LIN {X 0,Y 488.723,Z 208.607,A -85,B 0,C 180,E1 -6420.22,E2 -6420.22} C_VEL
LIN {X 0,Y 488.715,Z 208.607,A -85,B 0,C 180,E1 -6423.48,E2 -6423.48} C_VEL
LIN {X 0,Y 488.671,Z 208.616,A -85,B 0,C 180,E1 -6426.352,E2 -6426.352} C_VEL
LIN {X 0,Y 488.676,Z 208.612,A -85,B 0,C 180,E1 -6429.258,E2 -6429.258} C_VEL
LIN {X 0,Y 488.654,Z 208.617,A -85,B 0,C 180,E1 -6432.531,E2 -6432.531} C_VEL
LIN {X 0,Y 488.702,Z 208.608,A -85,B 0,C 180,E1 -6435.197,E2 -6435.197} C_VEL
LIN {X 0,Y 488.648,Z 208.619,A -85,B 0,C 180,E1 -6438.578,E2 -6438.578} C_VEL
LIN {X 0,Y 488.646,Z 208.619,A -85,B 0,C 180,E1 -6441.796,E2 -6441.796} C_VEL
LIN {X 0,Y 488.678,Z 208.611,A -85,B 0,C 180,E1 -6445.061,E2 -6445.061} C_VEL
LIN {X 0,Y 488.695,Z 208.612,A -85,B 0,C 180,E1 -6448.049,E2 -6448.049} C_VEL
LIN {X 0,Y 488.667,Z 208.614,A -85,B 0,C 180,E1 -6451.32,E2 -6451.32} C_VEL
LIN {X 0,Y 488.674,Z 208.616,A -85,B 0,C 180,E1 -6453.523,E2 -6453.523} C_VEL
LIN {X 0,Y 488.675,Z 208.614,A -85,B 0,C 180,E1 -6456.253,E2 -6456.253} C_VEL
LIN {X 0,Y 488.77,Z 208.751,A -85,B 0,C 180,E1 -6459.236,E2 -6459.236} C_VEL
LIN {X 0,Y 489.525,Z 214.415,A -85,B 0,C 180,E1 -6460.5,E2 -6460.5} C_VEL
LIN {X 0,Y 489.3,Z 225.378,A -85,B 0,C 180,E1 -6462.843,E2 -6462.843} C_VEL
LIN {X 0,Y 491.728,Z 238.426,A -85,B 0,C 180,E1 -6463.139,E2 -6463.139} C_VEL
LIN {X 0,Y 490.807,Z 332.574,A -85,B 0,C 180,E1 -6464.665,E2 -6464.665} C_VEL
LIN {X 0,Y 490.602,Z 346.158,A -85,B 0,C 180,E1 -6465.057,E2 -6465.057} C_VEL
LIN {X 0,Y 490.356,Z 358.525,A -85,B 0,C 180,E1 -6465.58,E2 -6465.58} C_VEL
LIN {X 0,Y 489.939,Z 371.206,A -85,B 0,C 180,E1 -6466.309,E2 -6466.309} C_VEL
LIN {X 0,Y 489.583,Z 382.52,A -85,B 0,C 180,E1 -6467.144,E2 -6467.144} C_VEL
LIN {X 0,Y 489.305,Z 392.196,A -85,B 0,C 180,E1 -6468.033,E2 -6468.033} C_VEL
LIN {X 0,Y 488.976,Z 401.025,A -85,B 0,C 180,E1 -6469.021,E2 -6469.021} C_VEL
LIN {X 0,Y 488.645,Z 410.097,A -85,B 0,C 180,E1 -6470.27,E2 -6470.27} C_VEL
LIN {X 0,Y 488.399,Z 417.387,A -85,B 0,C 180,E1 -6471.518,E2 -6471.518} C_VEL
LIN {X 0,Y 488.261,Z 422.294,A -85,B 0,C 180,E1 -6472.556,E2 -6472.556} C_VEL
LIN {X 0,Y 488.159,Z 426.656,A -85,B 0,C 180,E1 -6473.689,E2 -6473.689} C_VEL
LIN {X 0,Y 487.975,Z 430.671,A -85,B 0,C 180,E1 -6475.042,E2 -6475.042} C_VEL
LIN {X 0,Y 488.049,Z 432.509,A -85,B 0,C 180,E1 -6475.871,E2 -6475.871} C_VEL
LIN {X 0,Y 488.018,Z 433.894,A -85,B 0,C 180,E1 -6476.697,E2 -6476.697} C_VEL
LIN {X 0,Y 488.001,Z 434.882,A -85,B 0,C 180,E1 -6477.524,E2 -6477.524} C_VEL
LIN {X 0,Y 487.897,Z 435.478,A -85,B 0,C 180,E1 -6478.349,E2 -6478.349} C_VEL
LIN {X 0,Y 487.846,Z 435.628,A -85,B 0,C 180,E1 -6479.174,E2 -6479.174} C_VEL
LIN {X 0,Y 487.853,Z 434.72,A -85,B 0,C 180,E1 -6480.825,E2 -6480.825} C_VEL
LIN {X 0,Y 487.906,Z 433.666,A -85,B 0,C 180,E1 -6481.651,E2 -6481.651} C_VEL
LIN {X 0,Y 488.031,Z 432.145,A -85,B 0,C 180,E1 -6482.476,E2 -6482.476} C_VEL
LIN {X 0,Y 488.153,Z 429.067,A -85,B 0,C 180,E1 -6483.714,E2 -6483.714} C_VEL
LIN {X 0,Y 488.245,Z 424.918,A -85,B 0,C 180,E1 -6484.954,E2 -6484.954} C_VEL
LIN {X 0,Y 488.423,Z 419.571,A -85,B 0,C 180,E1 -6486.195,E2 -6486.195} C_VEL
LIN {X 0,Y 488.576,Z 412.853,A -85,B 0,C 180,E1 -6487.438,E2 -6487.438} C_VEL
LIN {X 0,Y 488.874,Z 404.478,A -85,B 0,C 180,E1 -6488.682,E2 -6488.682} C_VEL
LIN {X 0,Y 489.2,Z 395.816,A -85,B 0,C 180,E1 -6489.718,E2 -6489.718} C_VEL
LIN {X 0,Y 489.533,Z 385.151,A -85,B 0,C 180,E1 -6490.756,E2 -6490.756} C_VEL
LIN {X 0,Y 489.943,Z 374.542,A -85,B 0,C 180,E1 -6491.585,E2 -6491.585} C_VEL
LIN {X 0,Y 490.244,Z 362.686,A -85,B 0,C 180,E1 -6492.312,E2 -6492.312} C_VEL
LIN {X 0,Y 490.576,Z 349.695,A -85,B 0,C 180,E1 -6492.912,E2 -6492.912} C_VEL
LIN {X 0,Y 490.694,Z 337.931,A -85,B 0,C 180,E1 -6493.3,E2 -6493.3} C_VEL
LIN {X 0,Y 490.842,Z 323.698,A -85,B 0,C 180,E1 -6493.586,E2 -6493.586} C_VEL
LIN {X 0,Y 491.861,Z 237.927,A -85,B 0,C 180,E1 -6495.023,E2 -6495.023} C_VEL
LIN {X 0,Y 489.611,Z 227.078,A -85,B 0,C 180,E1 -6495.32,E2 -6495.32} C_VEL
LIN {X 0,Y 490.002,Z 217.222,A -85,B 0,C 180,E1 -6497.53,E2 -6497.53} C_VEL
LIN {X 0,Y 489.355,Z 211.542,A -85,B 0,C 180,E1 -6498.888,E2 -6498.888} C_VEL
LIN {X 0,Y 488.757,Z 208.607,A -85,B 0,C 180,E1 -6499.64,E2 -6499.64} C_VEL
LIN {X 0,Y 488.727,Z 208.609,A -85,B 0,C 180,E1 -6502.847,E2 -6502.847} C_VEL
LIN {X 0,Y 488.732,Z 208.607,A -85,B 0,C 180,E1 -6505.557,E2 -6505.557} C_VEL
LIN {X 0,Y 488.749,Z 208.608,A -85,B 0,C 180,E1 -6508.328,E2 -6508.328} C_VEL
LIN {X 0,Y 488.696,Z 208.609,A -85,B 0,C 180,E1 -6511.179,E2 -6511.179} C_VEL
LIN {X 0,Y 488.736,Z 208.608,A -85,B 0,C 180,E1 -6514.112,E2 -6514.112} C_VEL
LIN {X 0,Y 488.684,Z 208.61,A -85,B 0,C 180,E1 -6517.159,E2 -6517.159} C_VEL
LIN {X 0,Y 488.723,Z 208.609,A -85,B 0,C 180,E1 -6520.344,E2 -6520.344} C_VEL
LIN {X 0,Y 488.689,Z 208.612,A -85,B 0,C 180,E1 -6523.654,E2 -6523.654} C_VEL
LIN {X 0,Y 488.683,Z 208.614,A -85,B 0,C 180,E1 -6526.344,E2 -6526.344} C_VEL
LIN {X 0,Y 488.708,Z 208.611,A -85,B 0,C 180,E1 -6529.673,E2 -6529.673} C_VEL
LIN {X 0,Y 488.675,Z 208.612,A -85,B 0,C 180,E1 -6532.84,E2 -6532.84} C_VEL
LIN {X 0,Y 488.735,Z 208.61,A -85,B 0,C 180,E1 -6535.887,E2 -6535.887} C_VEL
LIN {X 0,Y 488.697,Z 208.614,A -85,B 0,C 180,E1 -6538.82,E2 -6538.82} C_VEL
LIN {X 0,Y 488.716,Z 208.616,A -85,B 0,C 180,E1 -6541.669,E2 -6541.669} C_VEL
LIN {X 0,Y 488.748,Z 208.686,A -85,B 0,C 180,E1 -6543.871,E2 -6543.871} C_VEL
LIN {X 0,Y 490.688,Z 218.243,A -85,B 0,C 180,E1 -6545.682,E2 -6545.682} C_VEL
LIN {X 0,Y 490.806,Z 223.126,A -85,B 0,C 180,E1 -6546.539,E2 -6546.539} C_VEL
LIN {X 0,Y 490.103,Z 239.074,A -85,B 0,C 180,E1 -6549.211,E2 -6549.211} C_VEL
LIN {X 0,Y 489.482,Z 257.613,A -85,B 0,C 180,E1 -6552.234,E2 -6552.234} C_VEL
LIN {X 0,Y 489.2,Z 266.659,A -85,B 0,C 180,E1 -6553.687,E2 -6553.687} C_VEL
LIN {X 0,Y 491.59,Z 284.59,A -85,B 0,C 180,E1 -6554.091,E2 -6554.091} C_VEL
LIN {X 0,Y 490.631,Z 377.059,A -85,B 0,C 180,E1 -6555.64,E2 -6555.64} C_VEL
LIN {X 0,Y 490.339,Z 391.13,A -85,B 0,C 180,E1 -6556.055,E2 -6556.055} C_VEL
LIN {X 0,Y 489.975,Z 404.148,A -85,B 0,C 180,E1 -6556.626,E2 -6556.626} C_VEL
LIN {X 0,Y 489.605,Z 416.588,A -85,B 0,C 180,E1 -6557.355,E2 -6557.355} C_VEL
LIN {X 0,Y 489.179,Z 427.818,A -85,B 0,C 180,E1 -6558.196,E2 -6558.196} C_VEL
LIN {X 0,Y 488.867,Z 438.762,A -85,B 0,C 180,E1 -6559.228,E2 -6559.228} C_VEL
LIN {X 0,Y 488.503,Z 447.75,A -85,B 0,C 180,E1 -6560.267,E2 -6560.267} C_VEL
LIN {X 0,Y 488.3,Z 456.482,A -85,B 0,C 180,E1 -6561.516,E2 -6561.516} C_VEL
LIN {X 0,Y 488.115,Z 463.485,A -85,B 0,C 180,E1 -6562.761,E2 -6562.761} C_VEL
LIN {X 0,Y 488.008,Z 469.913,A -85,B 0,C 180,E1 -6564.213,E2 -6564.213} C_VEL
LIN {X 0,Y 487.921,Z 474.083,A -85,B 0,C 180,E1 -6565.455,E2 -6565.455} C_VEL
LIN {X 0,Y 487.969,Z 477.17,A -85,B 0,C 180,E1 -6566.696,E2 -6566.696} C_VEL
LIN {X 0,Y 487.933,Z 478.647,A -85,B 0,C 180,E1 -6567.523,E2 -6567.523} C_VEL
LIN {X 0,Y 487.892,Z 479.698,A -85,B 0,C 180,E1 -6568.348,E2 -6568.348} C_VEL
LIN {X 0,Y 487.839,Z 480.346,A -85,B 0,C 180,E1 -6569.174,E2 -6569.174} C_VEL
LIN {X 0,Y 487.829,Z 480.588,A -85,B 0,C 180,E1 -6569.999,E2 -6569.999} C_VEL
LIN {X 0,Y 487.839,Z 480.378,A -85,B 0,C 180,E1 -6570.825,E2 -6570.825} C_VEL
LIN {X 0,Y 487.892,Z 479.765,A -85,B 0,C 180,E1 -6571.65,E2 -6571.65} C_VEL
LIN {X 0,Y 487.933,Z 478.75,A -85,B 0,C 180,E1 -6572.476,E2 -6572.476} C_VEL
LIN {X 0,Y 487.968,Z 477.306,A -85,B 0,C 180,E1 -6573.302,E2 -6573.302} C_VEL
LIN {X 0,Y 487.919,Z 474.284,A -85,B 0,C 180,E1 -6574.543,E2 -6574.543} C_VEL
LIN {X 0,Y 488.001,Z 470.186,A -85,B 0,C 180,E1 -6575.785,E2 -6575.785} C_VEL
LIN {X 0,Y 488.171,Z 463.861,A -85,B 0,C 180,E1 -6577.236,E2 -6577.236} C_VEL
LIN {X 0,Y 488.301,Z 456.957,A -85,B 0,C 180,E1 -6578.483,E2 -6578.483} C_VEL
LIN {X 0,Y 488.528,Z 448.344,A -85,B 0,C 180,E1 -6579.731,E2 -6579.731} C_VEL
LIN {X 0,Y 488.853,Z 439.479,A -85,B 0,C 180,E1 -6580.771,E2 -6580.771} C_VEL
LIN {X 0,Y 489.221,Z 428.764,A -85,B 0,C 180,E1 -6581.794,E2 -6581.794} C_VEL
LIN {X 0,Y 489.581,Z 417.955,A -85,B 0,C 180,E1 -6582.623,E2 -6582.623} C_VEL
LIN {X 0,Y 490.005,Z 405.415,A -85,B 0,C 180,E1 -6583.371,E2 -6583.371} C_VEL
LIN {X 0,Y 490.327,Z 392.679,A -85,B 0,C 180,E1 -6583.943,E2 -6583.943} C_VEL
LIN {X 0,Y 490.73,Z 380.124,A -85,B 0,C 180,E1 -6584.328,E2 -6584.328} C_VEL
LIN {X 0,Y 490.899,Z 363.057,A -85,B 0,C 180,E1 -6584.641,E2 -6584.641} C_VEL
LIN {X 0,Y 491.485,Z 283.418,A -85,B 0,C 180,E1 -6585.92,E2 -6585.92} C_VEL
LIN {X 0,Y 489.262,Z 267.955,A -85,B 0,C 180,E1 -6586.266,E2 -6586.266} C_VEL
LIN {X 0,Y 489.868,Z 249.29,A -85,B 0,C 180,E1 -6589.266,E2 -6589.266} C_VEL
LIN {X 0,Y 490.552,Z 230.601,A -85,B 0,C 180,E1 -6592.311,E2 -6592.311} C_VEL
LIN {X 0,Y 490.952,Z 219.899,A -85,B 0,C 180,E1 -6594.077,E2 -6594.077} C_VEL
LIN {X 0,Y 488.78,Z 208.604,A -85,B 0,C 180,E1 -6596.125,E2 -6596.125} C_VEL
LIN {X 0,Y 488.719,Z 208.607,A -85,B 0,C 180,E1 -6599.269,E2 -6599.269} C_VEL
LIN {X 0,Y 488.7,Z 208.603,A -85,B 0,C 180,E1 -6602.146,E2 -6602.146} C_VEL
LIN {X 0,Y 488.712,Z 208.6,A -85,B 0,C 180,E1 -6605.114,E2 -6605.114} C_VEL
LIN {X 0,Y 488.67,Z 208.61,A -85,B 0,C 180,E1 -6608.2,E2 -6608.2} C_VEL
LIN {X 0,Y 488.675,Z 208.615,A -85,B 0,C 180,E1 -6611.418,E2 -6611.418} C_VEL
LIN {X 0,Y 488.695,Z 208.606,A -85,B 0,C 180,E1 -6614.802,E2 -6614.802} C_VEL
LIN {X 0,Y 488.66,Z 208.613,A -85,B 0,C 180,E1 -6617.471,E2 -6617.471} C_VEL
LIN {X 0,Y 488.686,Z 208.608,A -85,B 0,C 180,E1 -6620.744,E2 -6620.744} C_VEL
LIN {X 0,Y 488.669,Z 208.603,A -85,B 0,C 180,E1 -6623.867,E2 -6623.867} C_VEL
LIN {X 0,Y 488.727,Z 208.604,A -85,B 0,C 180,E1 -6626.876,E2 -6626.876} C_VEL
LIN {X 0,Y 488.707,Z 208.597,A -85,B 0,C 180,E1 -6629.78,E2 -6629.78} C_VEL
LIN {X 0,Y 488.689,Z 208.611,A -85,B 0,C 180,E1 -6633.078,E2 -6633.078} C_VEL
LIN {X 0,Y 488.659,Z 208.608,A -85,B 0,C 180,E1 -6636.253,E2 -6636.253} C_VEL
LIN {X 0,Y 488.737,Z 208.601,A -85,B 0,C 180,E1 -6639.176,E2 -6639.176} C_VEL
LIN {X 0,Y 488.688,Z 208.61,A -85,B 0,C 180,E1 -6642.422,E2 -6642.422} C_VEL
LIN {X 0,Y 488.741,Z 208.594,A -85,B 0,C 180,E1 -6644.999,E2 -6644.999} C_VEL
LIN {X 0,Y 488.794,Z 208.594,A -85,B 0,C 180,E1 -6648.387,E2 -6648.387} C_VEL
LIN {X 0,Y 488.768,Z 208.597,A -85,B 0,C 180,E1 -6651.733,E2 -6651.733} C_VEL
LIN {X 0,Y 488.795,Z 208.589,A -85,B 0,C 180,E1 -6654.224,E2 -6654.224} C_VEL
LIN {X 0,Y 488.94,Z 208.574,A -85,B 0,C 180,E1 -6657.529,E2 -6657.529} C_VEL
LIN {X 0,Y 488.903,Z 208.576,A -85,B 0,C 180,E1 -6660.824,E2 -6660.824} C_VEL
LIN {X 0,Y 488.94,Z 208.568,A -85,B 0,C 180,E1 -6662.472,E2 -6662.472} C_VEL
LIN {X 0,Y 488.837,Z 208.589,A -85,B 0,C 180,E1 -6665.776,E2 -6665.776} C_VEL
LIN {X 0,Y 488.806,Z 208.592,A -85,B 0,C 180,E1 -6668.267,E2 -6668.267} C_VEL
LIN {X 0,Y 488.797,Z 208.589,A -85,B 0,C 180,E1 -6671.613,E2 -6671.613} C_VEL
LIN {X 0,Y 488.754,Z 208.598,A -85,B 0,C 180,E1 -6675.001,E2 -6675.001} C_VEL
LIN {X 0,Y 488.739,Z 208.598,A -85,B 0,C 180,E1 -6678.443,E2 -6678.443} C_VEL
LIN {X 0,Y 488.7,Z 208.608,A -85,B 0,C 180,E1 -6681.071,E2 -6681.071} C_VEL
LIN {X 0,Y 488.686,Z 208.607,A -85,B 0,C 180,E1 -6683.746,E2 -6683.746} C_VEL
LIN {X 0,Y 488.784,Z 208.598,A -85,B 0,C 180,E1 -6686.944,E2 -6686.944} C_VEL
LIN {X 0,Y 488.704,Z 208.604,A -85,B 0,C 180,E1 -6690.364,E2 -6690.364} C_VEL
LIN {X 0,Y 488.73,Z 208.604,A -85,B 0,C 180,E1 -6693.485,E2 -6693.485} C_VEL
LIN {X 0,Y 488.683,Z 208.611,A -85,B 0,C 180,E1 -6696.356,E2 -6696.356} C_VEL
LIN {X 0,Y 488.697,Z 208.614,A -85,B 0,C 180,E1 -6699.255,E2 -6699.255} C_VEL
LIN {X 0,Y 488.704,Z 208.606,A -85,B 0,C 180,E1 -6701.601,E2 -6701.601} C_VEL
LIN {X 0,Y 488.709,Z 208.611,A -85,B 0,C 180,E1 -6704.802,E2 -6704.802} C_VEL
LIN {X 0,Y 488.689,Z 208.609,A -85,B 0,C 180,E1 -6707.476,E2 -6707.476} C_VEL
LIN {X 0,Y 488.731,Z 208.602,A -85,B 0,C 180,E1 -6709.678,E2 -6709.678} C_VEL
LIN {X 0,Y 488.678,Z 208.616,A -85,B 0,C 180,E1 -6712.842,E2 -6712.842} C_VEL
LIN {X 0,Y 488.733,Z 208.606,A -85,B 0,C 180,E1 -6715.889,E2 -6715.889} C_VEL
LIN {X 0,Y 488.782,Z 208.621,A -85,B 0,C 180,E1 -6718.064,E2 -6718.064} C_VEL
LIN {X 0,Y 489.044,Z 221.936,A -85,B 0,C 180,E1 -6719.712,E2 -6719.712} C_VEL
LIN {X 0,Y 491.825,Z 237.317,A -85,B 0,C 180,E1 -6720.053,E2 -6720.053} C_VEL
LIN {X 0,Y 491.789,Z 246.688,A -85,B 0,C 180,E1 -6720.193,E2 -6720.193} C_VEL
LIN {X 0,Y 491.066,Z 252.538,A -85,B 0,C 180,E1 -6720.255,E2 -6720.255} C_VEL
LIN {X 0,Y 485.39,Z 271.547,A -85,B 0,C 180,E1 -6720.34,E2 -6720.34} C_VEL
LIN {X 0,Y 484.784,Z 277.391,A -85,B 0,C 180,E1 -6720.408,E2 -6720.408} C_VEL
LIN {X 0,Y 484.329,Z 332.155,A -85,B 0,C 180,E1 -6721.242,E2 -6721.242} C_VEL
LIN {X 0,Y 484.084,Z 345.66,A -85,B 0,C 180,E1 -6721.611,E2 -6721.611} C_VEL
LIN {X 0,Y 483.812,Z 357.944,A -85,B 0,C 180,E1 -6722.125,E2 -6722.125} C_VEL
LIN {X 0,Y 483.449,Z 369.727,A -85,B 0,C 180,E1 -6722.787,E2 -6722.787} C_VEL
LIN {X 0,Y 483.011,Z 380.235,A -85,B 0,C 180,E1 -6723.539,E2 -6723.539} C_VEL
LIN {X 0,Y 482.603,Z 389.782,A -85,B 0,C 180,E1 -6724.384,E2 -6724.384} C_VEL
LIN {X 0,Y 482.225,Z 399.602,A -85,B 0,C 180,E1 -6725.459,E2 -6725.459} C_VEL
LIN {X 0,Y 481.837,Z 408.121,A -85,B 0,C 180,E1 -6726.604,E2 -6726.604} C_VEL
LIN {X 0,Y 481.49,Z 416.045,A -85,B 0,C 180,E1 -6727.924,E2 -6727.924} C_VEL
LIN {X 0,Y 481.25,Z 422.003,A -85,B 0,C 180,E1 -6729.17,E2 -6729.17} C_VEL
LIN {X 0,Y 481.061,Z 426.585,A -85,B 0,C 180,E1 -6730.367,E2 -6730.367} C_VEL
LIN {X 0,Y 480.974,Z 430.659,A -85,B 0,C 180,E1 -6731.767,E2 -6731.767} C_VEL
LIN {X 0,Y 480.818,Z 433.245,A -85,B 0,C 180,E1 -6733.003,E2 -6733.003} C_VEL
LIN {X 0,Y 480.773,Z 434.526,A -85,B 0,C 180,E1 -6733.875,E2 -6733.875} C_VEL
LIN {X 0,Y 480.791,Z 435.38,A -85,B 0,C 180,E1 -6734.746,E2 -6734.746} C_VEL
LIN {X 0,Y 480.778,Z 435.771,A -85,B 0,C 180,E1 -6735.612,E2 -6735.612} C_VEL
LIN {X 0,Y 480.753,Z 435.765,A -85,B 0,C 180,E1 -6736.474,E2 -6736.474} C_VEL
LIN {X 0,Y 480.776,Z 435.361,A -85,B 0,C 180,E1 -6737.335,E2 -6737.335} C_VEL
LIN {X 0,Y 480.847,Z 434.345,A -85,B 0,C 180,E1 -6738.314,E2 -6738.314} C_VEL
LIN {X 0,Y 480.906,Z 431.581,A -85,B 0,C 180,E1 -6739.901,E2 -6739.901} C_VEL
LIN {X 0,Y 481.007,Z 428.224,A -85,B 0,C 180,E1 -6741.176,E2 -6741.176} C_VEL
LIN {X 0,Y 481.174,Z 423.786,A -85,B 0,C 180,E1 -6742.447,E2 -6742.447} C_VEL
LIN {X 0,Y 481.388,Z 417.051,A -85,B 0,C 180,E1 -6743.925,E2 -6743.925} C_VEL
LIN {X 0,Y 481.712,Z 409.761,A -85,B 0,C 180,E1 -6745.189,E2 -6745.189} C_VEL
LIN {X 0,Y 481.991,Z 402.345,A -85,B 0,C 180,E1 -6746.239,E2 -6746.239} C_VEL
LIN {X 0,Y 482.43,Z 392.313,A -85,B 0,C 180,E1 -6747.392,E2 -6747.392} C_VEL
LIN {X 0,Y 482.82,Z 382.19,A -85,B 0,C 180,E1 -6748.333,E2 -6748.333} C_VEL
LIN {X 0,Y 483.303,Z 370.932,A -85,B 0,C 180,E1 -6749.168,E2 -6749.168} C_VEL
LIN {X 0,Y 483.676,Z 358.102,A -85,B 0,C 180,E1 -6749.897,E2 -6749.897} C_VEL
LIN {X 0,Y 483.981,Z 345.669,A -85,B 0,C 180,E1 -6750.417,E2 -6750.417} C_VEL
LIN {X 0,Y 484.228,Z 332.434,A -85,B 0,C 180,E1 -6750.781,E2 -6750.781} C_VEL
LIN {X 0,Y 484.882,Z 237.942,A -85,B 0,C 180,E1 -6752.207,E2 -6752.207} C_VEL
LIN {X 0,Y 482,Z 221.981,A -85,B 0,C 180,E1 -6752.56,E2 -6752.56} C_VEL
LIN {X 0,Y 481.674,Z 209.489,A -85,B 0,C 180,E1 -6754.132,E2 -6754.132} C_VEL
LIN {X 0,Y 481.773,Z 209.472,A -85,B 0,C 180,E1 -6756.703,E2 -6756.703} C_VEL
LIN {X 0,Y 481.734,Z 209.48,A -85,B 0,C 180,E1 -6759.236,E2 -6759.236} C_VEL
LIN {X 0,Y 481.76,Z 209.473,A -85,B 0,C 180,E1 -6762.2,E2 -6762.2} C_VEL
LIN {X 0,Y 481.731,Z 209.479,A -85,B 0,C 180,E1 -6765.659,E2 -6765.659} C_VEL
LIN {X 0,Y 481.714,Z 209.482,A -85,B 0,C 180,E1 -6768.722,E2 -6768.722} C_VEL
LIN {X 0,Y 481.652,Z 209.489,A -85,B 0,C 180,E1 -6771.395,E2 -6771.395} C_VEL
LIN {X 0,Y 481.654,Z 209.487,A -85,B 0,C 180,E1 -6774.115,E2 -6774.115} C_VEL
LIN {X 0,Y 481.658,Z 209.488,A -85,B 0,C 180,E1 -6777.117,E2 -6777.117} C_VEL
LIN {X 0,Y 481.672,Z 209.484,A -85,B 0,C 180,E1 -6779.742,E2 -6779.742} C_VEL
LIN {X 0,Y 481.657,Z 209.489,A -85,B 0,C 180,E1 -6782.676,E2 -6782.676} C_VEL
LIN {X 0,Y 481.632,Z 209.489,A -85,B 0,C 180,E1 -6785.711,E2 -6785.711} C_VEL
LIN {X 0,Y 481.628,Z 209.493,A -85,B 0,C 180,E1 -6788.864,E2 -6788.864} C_VEL
LIN {X 0,Y 481.615,Z 209.495,A -85,B 0,C 180,E1 -6792.165,E2 -6792.165} C_VEL
LIN {X 0,Y 481.656,Z 209.489,A -85,B 0,C 180,E1 -6794.459,E2 -6794.459} C_VEL
LIN {X 0,Y 481.617,Z 209.493,A -85,B 0,C 180,E1 -6796.856,E2 -6796.856} C_VEL
LIN {X 0,Y 481.633,Z 209.492,A -85,B 0,C 180,E1 -6800.055,E2 -6800.055} C_VEL
LIN {X 0,Y 481.602,Z 209.493,A -85,B 0,C 180,E1 -6803.25,E2 -6803.25} C_VEL
LIN {X 0,Y 481.677,Z 209.487,A -85,B 0,C 180,E1 -6806.327,E2 -6806.327} C_VEL
LIN {X 0,Y 481.624,Z 209.492,A -85,B 0,C 180,E1 -6809.424,E2 -6809.424} C_VEL
LIN {X 0,Y 481.647,Z 209.491,A -85,B 0,C 180,E1 -6812.164,E2 -6812.164} C_VEL
LIN {X 0,Y 481.675,Z 209.484,A -85,B 0,C 180,E1 -6814.967,E2 -6814.967} C_VEL
LIN {X 0,Y 481.654,Z 209.492,A -85,B 0,C 180,E1 -6817.705,E2 -6817.705} C_VEL
LIN {X 0,Y 481.694,Z 209.56,A -85,B 0,C 180,E1 -6819.08,E2 -6819.08} C_VEL
LIN {X 0,Y 482.542,Z 215.522,A -85,B 0,C 180,E1 -6820.428,E2 -6820.428} C_VEL
LIN {X 0,Y 482.34,Z 225.6,A -85,B 0,C 180,E1 -6822.607,E2 -6822.607} C_VEL
LIN {X 0,Y 484.848,Z 239.239,A -85,B 0,C 180,E1 -6822.931,E2 -6822.931} C_VEL
LIN {X 0,Y 483.897,Z 333.205,A -85,B 0,C 180,E1 -6824.494,E2 -6824.494} C_VEL
LIN {X 0,Y 483.683,Z 345.898,A -85,B 0,C 180,E1 -6824.865,E2 -6824.865} C_VEL
LIN {X 0,Y 483.433,Z 357.852,A -85,B 0,C 180,E1 -6825.369,E2 -6825.369} C_VEL
LIN {X 0,Y 483.095,Z 369.214,A -85,B 0,C 180,E1 -6826.003,E2 -6826.003} C_VEL
LIN {X 0,Y 482.655,Z 380.946,A -85,B 0,C 180,E1 -6826.849,E2 -6826.849} C_VEL
LIN {X 0,Y 482.309,Z 391.228,A -85,B 0,C 180,E1 -6827.774,E2 -6827.774} C_VEL
LIN {X 0,Y 482,Z 400.993,A -85,B 0,C 180,E1 -6828.86,E2 -6828.86} C_VEL
LIN {X 0,Y 481.646,Z 408.761,A -85,B 0,C 180,E1 -6829.915,E2 -6829.915} C_VEL
LIN {X 0,Y 481.413,Z 416.356,A -85,B 0,C 180,E1 -6831.182,E2 -6831.182} C_VEL
LIN {X 0,Y 481.197,Z 422.446,A -85,B 0,C 180,E1 -6832.447,E2 -6832.447} C_VEL
LIN {X 0,Y 481.094,Z 427.152,A -85,B 0,C 180,E1 -6833.682,E2 -6833.682} C_VEL
LIN {X 0,Y 480.91,Z 430.909,A -85,B 0,C 180,E1 -6834.969,E2 -6834.969} C_VEL
LIN {X 0,Y 480.953,Z 432.778,A -85,B 0,C 180,E1 -6835.81,E2 -6835.81} C_VEL
LIN {X 0,Y 480.944,Z 434.18,A -85,B 0,C 180,E1 -6836.649,E2 -6836.649} C_VEL
LIN {X 0,Y 480.909,Z 435.182,A -85,B 0,C 180,E1 -6837.487,E2 -6837.487} C_VEL
LIN {X 0,Y 480.829,Z 435.792,A -85,B 0,C 180,E1 -6838.325,E2 -6838.325} C_VEL
LIN {X 0,Y 480.772,Z 435.962,A -85,B 0,C 180,E1 -6839.162,E2 -6839.162} C_VEL
LIN {X 0,Y 480.778,Z 435.073,A -85,B 0,C 180,E1 -6840.837,E2 -6840.837} C_VEL
LIN {X 0,Y 480.838,Z 434.029,A -85,B 0,C 180,E1 -6841.675,E2 -6841.675} C_VEL
LIN {X 0,Y 480.971,Z 432.517,A -85,B 0,C 180,E1 -6842.512,E2 -6842.512} C_VEL
LIN {X 0,Y 481.076,Z 429.45,A -85,B 0,C 180,E1 -6843.769,E2 -6843.769} C_VEL
LIN {X 0,Y 481.182,Z 425.303,A -85,B 0,C 180,E1 -6845.027,E2 -6845.027} C_VEL
LIN {X 0,Y 481.39,Z 419.958,A -85,B 0,C 180,E1 -6846.286,E2 -6846.286} C_VEL
LIN {X 0,Y 481.551,Z 413.25,A -85,B 0,C 180,E1 -6847.547,E2 -6847.547} C_VEL
LIN {X 0,Y 481.864,Z 404.888,A -85,B 0,C 180,E1 -6848.809,E2 -6848.809} C_VEL
LIN {X 0,Y 482.211,Z 396.243,A -85,B 0,C 180,E1 -6849.86,E2 -6849.86} C_VEL
LIN {X 0,Y 482.573,Z 385.583,A -85,B 0,C 180,E1 -6850.913,E2 -6850.913} C_VEL
LIN {X 0,Y 483.014,Z 374.993,A -85,B 0,C 180,E1 -6851.754,E2 -6851.754} C_VEL
LIN {X 0,Y 483.328,Z 363.194,A -85,B 0,C 180,E1 -6852.491,E2 -6852.491} C_VEL
LIN {X 0,Y 483.703,Z 349.765,A -85,B 0,C 180,E1 -6853.121,E2 -6853.121} C_VEL
LIN {X 0,Y 483.838,Z 337.706,A -85,B 0,C 180,E1 -6853.519,E2 -6853.519} C_VEL
LIN {X 0,Y 484.067,Z 321.685,A -85,B 0,C 180,E1 -6853.834,E2 -6853.834} C_VEL
LIN {X 0,Y 485.111,Z 238.965,A -85,B 0,C 180,E1 -6855.265,E2 -6855.265} C_VEL
LIN {X 0,Y 482.71,Z 227.523,A -85,B 0,C 180,E1 -6855.594,E2 -6855.594} C_VEL
LIN {X 0,Y 483.071,Z 217.951,A -85,B 0,C 180,E1 -6857.789,E2 -6857.789} C_VEL
LIN {X 0,Y 482.311,Z 212.429,A -85,B 0,C 180,E1 -6859.138,E2 -6859.138} C_VEL
LIN {X 0,Y 481.695,Z 209.486,A -85,B 0,C 180,E1 -6859.94,E2 -6859.94} C_VEL
LIN {X 0,Y 481.67,Z 209.486,A -85,B 0,C 180,E1 -6863.201,E2 -6863.201} C_VEL
LIN {X 0,Y 481.694,Z 209.486,A -85,B 0,C 180,E1 -6865.957,E2 -6865.957} C_VEL
LIN {X 0,Y 481.704,Z 209.483,A -85,B 0,C 180,E1 -6868.781,E2 -6868.781} C_VEL
LIN {X 0,Y 481.662,Z 209.49,A -85,B 0,C 180,E1 -6872.189,E2 -6872.189} C_VEL
LIN {X 0,Y 481.694,Z 209.483,A -85,B 0,C 180,E1 -6874.682,E2 -6874.682} C_VEL
LIN {X 0,Y 481.66,Z 209.489,A -85,B 0,C 180,E1 -6878.007,E2 -6878.007} C_VEL
LIN {X 0,Y 481.661,Z 209.485,A -85,B 0,C 180,E1 -6881.041,E2 -6881.041} C_VEL
LIN {X 0,Y 481.66,Z 209.489,A -85,B 0,C 180,E1 -6884.457,E2 -6884.457} C_VEL
LIN {X 0,Y 481.648,Z 209.491,A -85,B 0,C 180,E1 -6887.838,E2 -6887.838} C_VEL
LIN {X 0,Y 481.664,Z 209.485,A -85,B 0,C 180,E1 -6890.654,E2 -6890.654} C_VEL
LIN {X 0,Y 481.626,Z 209.491,A -85,B 0,C 180,E1 -6893.377,E2 -6893.377} C_VEL
LIN {X 0,Y 481.715,Z 209.483,A -85,B 0,C 180,E1 -6896.329,E2 -6896.329} C_VEL
LIN {X 0,Y 481.655,Z 209.494,A -85,B 0,C 180,E1 -6899.417,E2 -6899.417} C_VEL
LIN {X 0,Y 481.672,Z 209.492,A -85,B 0,C 180,E1 -6902.165,E2 -6902.165} C_VEL
LIN {X 0,Y 481.695,Z 209.556,A -85,B 0,C 180,E1 -6903.576,E2 -6903.576} C_VEL
LIN {X 0,Y 483.768,Z 219.614,A -85,B 0,C 180,E1 -6905.54,E2 -6905.54} C_VEL
LIN {X 0,Y 483.948,Z 223.948,A -85,B 0,C 180,E1 -6906.32,E2 -6906.32} C_VEL
LIN {X 0,Y 483.176,Z 240.339,A -85,B 0,C 180,E1 -6909.122,E2 -6909.122} C_VEL
LIN {X 0,Y 482.415,Z 260.085,A -85,B 0,C 180,E1 -6912.404,E2 -6912.404} C_VEL
LIN {X 0,Y 482.227,Z 266.197,A -85,B 0,C 180,E1 -6913.404,E2 -6913.404} C_VEL
LIN {X 0,Y 484.799,Z 285.359,A -85,B 0,C 180,E1 -6913.862,E2 -6913.862} C_VEL
LIN {X 0,Y 483.774,Z 376.435,A -85,B 0,C 180,E1 -6915.432,E2 -6915.432} C_VEL
LIN {X 0,Y 483.428,Z 390.507,A -85,B 0,C 180,E1 -6915.852,E2 -6915.852} C_VEL
LIN {X 0,Y 483.087,Z 402.598,A -85,B 0,C 180,E1 -6916.378,E2 -6916.378} C_VEL
LIN {X 0,Y 482.663,Z 414.443,A -85,B 0,C 180,E1 -6917.062,E2 -6917.062} C_VEL
LIN {X 0,Y 482.253,Z 426.565,A -85,B 0,C 180,E1 -6917.959,E2 -6917.959} C_VEL
LIN {X 0,Y 481.847,Z 437.278,A -85,B 0,C 180,E1 -6918.963,E2 -6918.963} C_VEL
LIN {X 0,Y 481.438,Z 447.29,A -85,B 0,C 180,E1 -6920.123,E2 -6920.123} C_VEL
LIN {X 0,Y 481.247,Z 454.74,A -85,B 0,C 180,E1 -6921.179,E2 -6921.179} C_VEL
LIN {X 0,Y 481.069,Z 462.042,A -85,B 0,C 180,E1 -6922.444,E2 -6922.444} C_VEL
LIN {X 0,Y 480.905,Z 468.407,A -85,B 0,C 180,E1 -6923.845,E2 -6923.845} C_VEL
LIN {X 0,Y 480.897,Z 472.432,A -85,B 0,C 180,E1 -6924.969,E2 -6924.969} C_VEL
LIN {X 0,Y 480.845,Z 474.848,A -85,B 0,C 180,E1 -6925.808,E2 -6925.808} C_VEL
LIN {X 0,Y 480.894,Z 476.824,A -85,B 0,C 180,E1 -6926.648,E2 -6926.648} C_VEL
LIN {X 0,Y 480.845,Z 478.308,A -85,B 0,C 180,E1 -6927.486,E2 -6927.486} C_VEL
LIN {X 0,Y 480.823,Z 479.366,A -85,B 0,C 180,E1 -6928.324,E2 -6928.324} C_VEL
LIN {X 0,Y 480.765,Z 480.019,A -85,B 0,C 180,E1 -6929.161,E2 -6929.161} C_VEL
LIN {X 0,Y 480.752,Z 480.262,A -85,B 0,C 180,E1 -6929.999,E2 -6929.999} C_VEL
LIN {X 0,Y 480.764,Z 480.051,A -85,B 0,C 180,E1 -6930.837,E2 -6930.837} C_VEL
LIN {X 0,Y 480.823,Z 479.436,A -85,B 0,C 180,E1 -6931.674,E2 -6931.674} C_VEL
LIN {X 0,Y 480.845,Z 478.416,A -85,B 0,C 180,E1 -6932.512,E2 -6932.512} C_VEL
LIN {X 0,Y 480.893,Z 476.962,A -85,B 0,C 180,E1 -6933.35,E2 -6933.35} C_VEL
LIN {X 0,Y 480.837,Z 473.925,A -85,B 0,C 180,E1 -6934.61,E2 -6934.61} C_VEL
LIN {X 0,Y 480.906,Z 469.806,A -85,B 0,C 180,E1 -6935.871,E2 -6935.871} C_VEL
LIN {X 0,Y 481.094,Z 463.453,A -85,B 0,C 180,E1 -6937.343,E2 -6937.343} C_VEL
LIN {X 0,Y 481.247,Z 456.52,A -85,B 0,C 180,E1 -6938.608,E2 -6938.608} C_VEL
LIN {X 0,Y 481.435,Z 449.437,A -85,B 0,C 180,E1 -6939.663,E2 -6939.663} C_VEL
LIN {X 0,Y 481.765,Z 440.907,A -85,B 0,C 180,E1 -6940.718,E2 -6940.718} C_VEL
LIN {X 0,Y 482.176,Z 430.355,A -85,B 0,C 180,E1 -6941.773,E2 -6941.773} C_VEL
LIN {X 0,Y 482.472,Z 419.91,A -85,B 0,C 180,E1 -6942.62,E2 -6942.62} C_VEL
LIN {X 0,Y 482.927,Z 408.519,A -85,B 0,C 180,E1 -6943.357,E2 -6943.357} C_VEL
LIN {X 0,Y 483.287,Z 396.887,A -85,B 0,C 180,E1 -6943.936,E2 -6943.936} C_VEL
LIN {X 0,Y 483.695,Z 383.676,A -85,B 0,C 180,E1 -6944.407,E2 -6944.407} C_VEL
LIN {X 0,Y 483.911,Z 371.096,A -85,B 0,C 180,E1 -6944.696,E2 -6944.696} C_VEL
LIN {X 0,Y 484.604,Z 284.104,A -85,B 0,C 180,E1 -6946.125,E2 -6946.125} C_VEL
LIN {X 0,Y 482.27,Z 267.79,A -85,B 0,C 180,E1 -6946.486,E2 -6946.486} C_VEL
LIN {X 0,Y 482.926,Z 248.966,A -85,B 0,C 180,E1 -6949.554,E2 -6949.554} C_VEL
LIN {X 0,Y 483.678,Z 230.275,A -85,B 0,C 180,E1 -6952.646,E2 -6952.646} C_VEL
LIN {X 0,Y 483.976,Z 220.92,A -85,B 0,C 180,E1 -6954.218,E2 -6954.218} C_VEL
LIN {X 0,Y 481.733,Z 209.482,A -85,B 0,C 180,E1 -6956.303,E2 -6956.303} C_VEL
LIN {X 0,Y 481.673,Z 209.484,A -85,B 0,C 180,E1 -6958.902,E2 -6958.902} C_VEL
LIN {X 0,Y 481.654,Z 209.48,A -85,B 0,C 180,E1 -6962.188,E2 -6962.188} C_VEL
LIN {X 0,Y 481.684,Z 209.475,A -85,B 0,C 180,E1 -6964.681,E2 -6964.681} C_VEL
LIN {X 0,Y 481.644,Z 209.487,A -85,B 0,C 180,E1 -6968.005,E2 -6968.005} C_VEL
LIN {X 0,Y 481.628,Z 209.489,A -85,B 0,C 180,E1 -6971.043,E2 -6971.043} C_VEL
LIN {X 0,Y 481.648,Z 209.484,A -85,B 0,C 180,E1 -6974.457,E2 -6974.457} C_VEL
LIN {X 0,Y 481.622,Z 209.484,A -85,B 0,C 180,E1 -6977.836,E2 -6977.836} C_VEL
LIN {X 0,Y 481.659,Z 209.488,A -85,B 0,C 180,E1 -6981.14,E2 -6981.14} C_VEL
LIN {X 0,Y 481.628,Z 209.477,A -85,B 0,C 180,E1 -6984.29,E2 -6984.29} C_VEL
LIN {X 0,Y 481.661,Z 209.488,A -85,B 0,C 180,E1 -6987.325,E2 -6987.325} C_VEL
LIN {X 0,Y 481.656,Z 209.474,A -85,B 0,C 180,E1 -6990.257,E2 -6990.257} C_VEL
LIN {X 0,Y 481.651,Z 209.488,A -85,B 0,C 180,E1 -6993.106,E2 -6993.106} C_VEL
LIN {X 0,Y 481.638,Z 209.481,A -85,B 0,C 180,E1 -6995.885,E2 -6995.885} C_VEL
LIN {X 0,Y 481.693,Z 209.475,A -85,B 0,C 180,E1 -6999.028,E2 -6999.028} C_VEL
LIN {X 0,Y 481.671,Z 209.482,A -85,B 0,C 180,E1 -7002.157,E2 -7002.157} C_VEL
LIN {X 0,Y 481.726,Z 209.47,A -85,B 0,C 180,E1 -7004.775,E2 -7004.775} C_VEL
LIN {X 0,Y 481.74,Z 209.471,A -85,B 0,C 180,E1 -7008.215,E2 -7008.215} C_VEL
LIN {X 0,Y 481.724,Z 209.474,A -85,B 0,C 180,E1 -7011.611,E2 -7011.611} C_VEL
LIN {X 0,Y 481.756,Z 209.466,A -85,B 0,C 180,E1 -7014.139,E2 -7014.139} C_VEL
LIN {X 0,Y 481.907,Z 209.45,A -85,B 0,C 180,E1 -7017.493,E2 -7017.493} C_VEL
LIN {X 0,Y 481.856,Z 209.454,A -85,B 0,C 180,E1 -7020.836,E2 -7020.836} C_VEL
LIN {X 0,Y 481.906,Z 209.443,A -85,B 0,C 180,E1 -7022.508,E2 -7022.508} C_VEL
LIN {X 0,Y 481.798,Z 209.467,A -85,B 0,C 180,E1 -7025.861,E2 -7025.861} C_VEL
LIN {X 0,Y 481.752,Z 209.469,A -85,B 0,C 180,E1 -7028.389,E2 -7028.389} C_VEL
LIN {X 0,Y 481.742,Z 209.469,A -85,B 0,C 180,E1 -7031.785,E2 -7031.785} C_VEL
LIN {X 0,Y 481.735,Z 209.474,A -85,B 0,C 180,E1 -7035.225,E2 -7035.225} C_VEL
LIN {X 0,Y 481.701,Z 209.474,A -85,B 0,C 180,E1 -7038.722,E2 -7038.722} C_VEL
LIN {X 0,Y 481.639,Z 209.491,A -85,B 0,C 180,E1 -7041.395,E2 -7041.395} C_VEL
LIN {X 0,Y 481.67,Z 209.479,A -85,B 0,C 180,E1 -7044.114,E2 -7044.114} C_VEL
LIN {X 0,Y 481.739,Z 209.478,A -85,B 0,C 180,E1 -7047.14,E2 -7047.14} C_VEL
LIN {X 0,Y 481.672,Z 209.484,A -85,B 0,C 180,E1 -7049.742,E2 -7049.742} C_VEL
LIN {X 0,Y 481.667,Z 209.484,A -85,B 0,C 180,E1 -7052.675,E2 -7052.675} C_VEL
LIN {X 0,Y 481.636,Z 209.491,A -85,B 0,C 180,E1 -7055.71,E2 -7055.71} C_VEL
LIN {X 0,Y 481.667,Z 209.484,A -85,B 0,C 180,E1 -7058.86,E2 -7058.86} C_VEL
LIN {X 0,Y 481.649,Z 209.483,A -85,B 0,C 180,E1 -7061.914,E2 -7061.914} C_VEL
LIN {X 0,Y 481.656,Z 209.487,A -85,B 0,C 180,E1 -7064.458,E2 -7064.458} C_VEL
LIN {X 0,Y 481.645,Z 209.485,A -85,B 0,C 180,E1 -7067.841,E2 -7067.841} C_VEL
LIN {X 0,Y 481.678,Z 209.487,A -85,B 0,C 180,E1 -7070.652,E2 -7070.652} C_VEL
LIN {X 0,Y 481.626,Z 209.491,A -85,B 0,C 180,E1 -7073.377,E2 -7073.377} C_VEL
LIN {X 0,Y 481.709,Z 209.484,A -85,B 0,C 180,E1 -7076.331,E2 -7076.331} C_VEL
LIN {X 0,Y 481.797,Z 209.632,A -85,B 0,C 180,E1 -7077.959,E2 -7077.959} C_VEL
LIN {X 0,Y 482.144,Z 222.241,A -85,B 0,C 180,E1 -7079.463,E2 -7079.463} C_VEL
LIN {X 0,Y 485.071,Z 238.895,A -85,B 0,C 180,E1 -7079.831,E2 -7079.831} C_VEL
LIN {X 0,Y 484.784,Z 277.391,A -85,B 0,C 180,E1 -7080.408,E2 -7080.408} C_VEL
LIN {X 0,Y 484.176,Z 283.235,A -85,B 0,C 180,E1 -7080.474,E2 -7080.474} C_VEL
LIN {X 0,Y 478.467,Z 302.24,A -85,B 0,C 180,E1 -7080.557,E2 -7080.557} C_VEL
LIN {X 0,Y 477.728,Z 308.09,A -85,B 0,C 180,E1 -7080.62,E2 -7080.62} C_VEL
LIN {X 0,Y 477.516,Z 334.294,A -85,B 0,C 180,E1 -7081.049,E2 -7081.049} C_VEL
LIN {X 0,Y 477.244,Z 346.632,A -85,B 0,C 180,E1 -7081.407,E2 -7081.407} C_VEL
LIN {X 0,Y 476.919,Z 359.641,A -85,B 0,C 180,E1 -7081.975,E2 -7081.975} C_VEL
LIN {X 0,Y 476.545,Z 372.051,A -85,B 0,C 180,E1 -7082.709,E2 -7082.709} C_VEL
LIN {X 0,Y 475.973,Z 383.499,A -85,B 0,C 180,E1 -7083.59,E2 -7083.59} C_VEL
LIN {X 0,Y 475.532,Z 394.167,A -85,B 0,C 180,E1 -7084.623,E2 -7084.623} C_VEL
LIN {X 0,Y 475.058,Z 403.607,A -85,B 0,C 180,E1 -7085.763,E2 -7085.763} C_VEL
LIN {X 0,Y 474.714,Z 411.54,A -85,B 0,C 180,E1 -7086.942,E2 -7086.942} C_VEL
LIN {X 0,Y 474.357,Z 418.743,A -85,B 0,C 180,E1 -7088.261,E2 -7088.261} C_VEL
LIN {X 0,Y 474.098,Z 424.566,A -85,B 0,C 180,E1 -7089.614,E2 -7089.614} C_VEL
LIN {X 0,Y 473.947,Z 429.045,A -85,B 0,C 180,E1 -7090.961,E2 -7090.961} C_VEL
LIN {X 0,Y 473.898,Z 431.374,A -85,B 0,C 180,E1 -7091.855,E2 -7091.855} C_VEL
LIN {X 0,Y 473.764,Z 433.226,A -85,B 0,C 180,E1 -7092.742,E2 -7092.742} C_VEL
LIN {X 0,Y 473.69,Z 434.583,A -85,B 0,C 180,E1 -7093.628,E2 -7093.628} C_VEL
LIN {X 0,Y 473.711,Z 435.654,A -85,B 0,C 180,E1 -7094.656,E2 -7094.656} C_VEL
LIN {X 0,Y 473.659,Z 436.117,A -85,B 0,C 180,E1 -7096.268,E2 -7096.268} C_VEL
LIN {X 0,Y 473.681,Z 435.787,A -85,B 0,C 180,E1 -7097.142,E2 -7097.142} C_VEL
LIN {X 0,Y 473.777,Z 434.764,A -85,B 0,C 180,E1 -7098.252,E2 -7098.252} C_VEL
LIN {X 0,Y 473.802,Z 432.297,A -85,B 0,C 180,E1 -7099.748,E2 -7099.748} C_VEL
LIN {X 0,Y 473.935,Z 429.089,A -85,B 0,C 180,E1 -7101.043,E2 -7101.043} C_VEL
LIN {X 0,Y 474.077,Z 424.821,A -85,B 0,C 180,E1 -7102.334,E2 -7102.334} C_VEL
LIN {X 0,Y 474.33,Z 418.802,A -85,B 0,C 180,E1 -7103.743,E2 -7103.743} C_VEL
LIN {X 0,Y 474.642,Z 411.262,A -85,B 0,C 180,E1 -7105.117,E2 -7105.117} C_VEL
LIN {X 0,Y 474.979,Z 402.511,A -85,B 0,C 180,E1 -7106.396,E2 -7106.396} C_VEL
LIN {X 0,Y 475.453,Z 392.432,A -85,B 0,C 180,E1 -7107.565,E2 -7107.565} C_VEL
LIN {X 0,Y 475.895,Z 382.259,A -85,B 0,C 180,E1 -7108.52,E2 -7108.52} C_VEL
LIN {X 0,Y 476.375,Z 370.926,A -85,B 0,C 180,E1 -7109.367,E2 -7109.367} C_VEL
LIN {X 0,Y 476.783,Z 358.004,A -85,B 0,C 180,E1 -7110.107,E2 -7110.107} C_VEL
LIN {X 0,Y 477.108,Z 345.345,A -85,B 0,C 180,E1 -7110.634,E2 -7110.634} C_VEL
LIN {X 0,Y 477.351,Z 331.75,A -85,B 0,C 180,E1 -7111.003,E2 -7111.003} C_VEL
LIN {X 0,Y 477.989,Z 238.537,A -85,B 0,C 180,E1 -7112.424,E2 -7112.424} C_VEL
LIN {X 0,Y 475.011,Z 222.081,A -85,B 0,C 180,E1 -7112.784,E2 -7112.784} C_VEL
LIN {X 0,Y 474.637,Z 210.365,A -85,B 0,C 180,E1 -7114.22,E2 -7114.22} C_VEL
LIN {X 0,Y 474.731,Z 210.35,A -85,B 0,C 180,E1 -7116.803,E2 -7116.803} C_VEL
LIN {X 0,Y 474.702,Z 210.355,A -85,B 0,C 180,E1 -7119.374,E2 -7119.374} C_VEL
LIN {X 0,Y 474.708,Z 210.352,A -85,B 0,C 180,E1 -7122.277,E2 -7122.277} C_VEL
LIN {X 0,Y 474.687,Z 210.356,A -85,B 0,C 180,E1 -7125.768,E2 -7125.768} C_VEL
LIN {X 0,Y 474.669,Z 210.359,A -85,B 0,C 180,E1 -7129.011,E2 -7129.011} C_VEL
LIN {X 0,Y 474.595,Z 210.366,A -85,B 0,C 180,E1 -7131.73,E2 -7131.73} C_VEL
LIN {X 0,Y 474.631,Z 210.364,A -85,B 0,C 180,E1 -7134.495,E2 -7134.495} C_VEL
LIN {X 0,Y 474.605,Z 210.367,A -85,B 0,C 180,E1 -7137.327,E2 -7137.327} C_VEL
LIN {X 0,Y 474.602,Z 210.367,A -85,B 0,C 180,E1 -7140.231,E2 -7140.231} C_VEL
LIN {X 0,Y 474.621,Z 210.364,A -85,B 0,C 180,E1 -7143.223,E2 -7143.223} C_VEL
LIN {X 0,Y 474.585,Z 210.371,A -85,B 0,C 180,E1 -7146.325,E2 -7146.325} C_VEL
LIN {X 0,Y 474.605,Z 210.365,A -85,B 0,C 180,E1 -7149.551,E2 -7149.551} C_VEL
LIN {X 0,Y 474.571,Z 210.371,A -85,B 0,C 180,E1 -7152.94,E2 -7152.94} C_VEL
LIN {X 0,Y 474.603,Z 210.368,A -85,B 0,C 180,E1 -7155.894,E2 -7155.894} C_VEL
LIN {X 0,Y 474.586,Z 210.367,A -85,B 0,C 180,E1 -7159.048,E2 -7159.048} C_VEL
LIN {X 0,Y 474.586,Z 210.37,A -85,B 0,C 180,E1 -7161.709,E2 -7161.709} C_VEL
LIN {X 0,Y 474.583,Z 210.368,A -85,B 0,C 180,E1 -7164.722,E2 -7164.722} C_VEL
LIN {X 0,Y 474.619,Z 210.366,A -85,B 0,C 180,E1 -7167.786,E2 -7167.786} C_VEL
LIN {X 0,Y 474.584,Z 210.367,A -85,B 0,C 180,E1 -7170.895,E2 -7170.895} C_VEL
LIN {X 0,Y 474.577,Z 210.371,A -85,B 0,C 180,E1 -7173.623,E2 -7173.623} C_VEL
LIN {X 0,Y 474.64,Z 210.36,A -85,B 0,C 180,E1 -7176.642,E2 -7176.642} C_VEL
LIN {X 0,Y 474.656,Z 210.415,A -85,B 0,C 180,E1 -7178.938,E2 -7178.938} C_VEL
LIN {X 0,Y 475.564,Z 216.597,A -85,B 0,C 180,E1 -7180.354,E2 -7180.354} C_VEL
LIN {X 0,Y 475.368,Z 225.903,A -85,B 0,C 180,E1 -7182.385,E2 -7182.385} C_VEL
LIN {X 0,Y 478.016,Z 239.901,A -85,B 0,C 180,E1 -7182.718,E2 -7182.718} C_VEL
LIN {X 0,Y 476.97,Z 333.741,A -85,B 0,C 180,E1 -7184.318,E2 -7184.318} C_VEL
LIN {X 0,Y 476.738,Z 347.078,A -85,B 0,C 180,E1 -7184.721,E2 -7184.721} C_VEL
LIN {X 0,Y 476.458,Z 359.327,A -85,B 0,C 180,E1 -7185.259,E2 -7185.259} C_VEL
LIN {X 0,Y 476.004,Z 371.964,A -85,B 0,C 180,E1 -7186.009,E2 -7186.009} C_VEL
LIN {X 0,Y 475.612,Z 383.264,A -85,B 0,C 180,E1 -7186.868,E2 -7186.868} C_VEL
LIN {X 0,Y 475.302,Z 392.711,A -85,B 0,C 180,E1 -7187.759,E2 -7187.759} C_VEL
LIN {X 0,Y 474.891,Z 402.593,A -85,B 0,C 180,E1 -7188.907,E2 -7188.907} C_VEL
LIN {X 0,Y 474.542,Z 411.536,A -85,B 0,C 180,E1 -7190.194,E2 -7190.194} C_VEL
LIN {X 0,Y 474.274,Z 418.652,A -85,B 0,C 180,E1 -7191.478,E2 -7191.478} C_VEL
LIN {X 0,Y 474.082,Z 424.333,A -85,B 0,C 180,E1 -7192.761,E2 -7192.761} C_VEL
LIN {X 0,Y 474.017,Z 428.781,A -85,B 0,C 180,E1 -7194.043,E2 -7194.043} C_VEL
LIN {X 0,Y 473.85,Z 431.137,A -85,B 0,C 180,E1 -7194.894,E2 -7194.894} C_VEL
LIN {X 0,Y 473.858,Z 433.038,A -85,B 0,C 180,E1 -7195.747,E2 -7195.747} C_VEL
LIN {X 0,Y 473.871,Z 434.46,A -85,B 0,C 180,E1 -7196.599,E2 -7196.599} C_VEL
LIN {X 0,Y 473.822,Z 435.48,A -85,B 0,C 180,E1 -7197.449,E2 -7197.449} C_VEL
LIN {X 0,Y 473.764,Z 436.105,A -85,B 0,C 180,E1 -7198.3,E2 -7198.3} C_VEL
LIN {X 0,Y 473.7,Z 436.298,A -85,B 0,C 180,E1 -7199.15,E2 -7199.15} C_VEL
LIN {X 0,Y 473.686,Z 436.062,A -85,B 0,C 180,E1 -7200,E2 -7200} C_VEL
LIN {X 0,Y 473.706,Z 435.43,A -85,B 0,C 180,E1 -7200.85,E2 -7200.85} C_VEL
LIN {X 0,Y 473.773,Z 434.398,A -85,B 0,C 180,E1 -7201.7,E2 -7201.7} C_VEL
LIN {X 0,Y 473.913,Z 432.9,A -85,B 0,C 180,E1 -7202.55,E2 -7202.55} C_VEL
LIN {X 0,Y 474.005,Z 429.849,A -85,B 0,C 180,E1 -7203.825,E2 -7203.825} C_VEL
LIN {X 0,Y 474.122,Z 425.716,A -85,B 0,C 180,E1 -7205.102,E2 -7205.102} C_VEL
LIN {X 0,Y 474.401,Z 419.368,A -85,B 0,C 180,E1 -7206.593,E2 -7206.593} C_VEL
LIN {X 0,Y 474.58,Z 412.436,A -85,B 0,C 180,E1 -7207.873,E2 -7207.873} C_VEL
LIN {X 0,Y 474.985,Z 403.712,A -85,B 0,C 180,E1 -7209.152,E2 -7209.152} C_VEL
LIN {X 0,Y 475.373,Z 393.785,A -85,B 0,C 180,E1 -7210.326,E2 -7210.326} C_VEL
LIN {X 0,Y 475.831,Z 383.661,A -85,B 0,C 180,E1 -7211.286,E2 -7211.286} C_VEL
LIN {X 0,Y 476.175,Z 374.004,A -85,B 0,C 180,E1 -7212.033,E2 -7212.033} C_VEL
LIN {X 0,Y 476.485,Z 361.848,A -85,B 0,C 180,E1 -7212.782,E2 -7212.782} C_VEL
LIN {X 0,Y 476.858,Z 349.031,A -85,B 0,C 180,E1 -7213.372,E2 -7213.372} C_VEL
LIN {X 0,Y 477.037,Z 336.62,A -85,B 0,C 180,E1 -7213.77,E2 -7213.77} C_VEL
LIN {X 0,Y 477.266,Z 317.03,A -85,B 0,C 180,E1 -7214.143,E2 -7214.143} C_VEL
LIN {X 0,Y 478.407,Z 240.119,A -85,B 0,C 180,E1 -7215.518,E2 -7215.518} C_VEL
LIN {X 0,Y 475.825,Z 228.052,A -85,B 0,C 180,E1 -7215.868,E2 -7215.868} C_VEL
LIN {X 0,Y 476.128,Z 218.689,A -85,B 0,C 180,E1 -7218.058,E2 -7218.058} C_VEL
LIN {X 0,Y 474.898,Z 211.462,A -85,B 0,C 180,E1 -7219.9,E2 -7219.9} C_VEL
LIN {X 0,Y 474.684,Z 210.361,A -85,B 0,C 180,E1 -7220.248,E2 -7220.248} C_VEL
LIN {X 0,Y 474.615,Z 210.365,A -85,B 0,C 180,E1 -7223.566,E2 -7223.566} C_VEL
LIN {X 0,Y 474.659,Z 210.363,A -85,B 0,C 180,E1 -7226.372,E2 -7226.372} C_VEL
LIN {X 0,Y 474.626,Z 210.363,A -85,B 0,C 180,E1 -7229.252,E2 -7229.252} C_VEL
LIN {X 0,Y 474.62,Z 210.367,A -85,B 0,C 180,E1 -7232.43,E2 -7232.43} C_VEL
LIN {X 0,Y 474.62,Z 210.363,A -85,B 0,C 180,E1 -7235.469,E2 -7235.469} C_VEL
LIN {X 0,Y 474.616,Z 210.366,A -85,B 0,C 180,E1 -7238.457,E2 -7238.457} C_VEL
LIN {X 0,Y 474.632,Z 210.36,A -85,B 0,C 180,E1 -7240.959,E2 -7240.959} C_VEL
LIN {X 0,Y 474.61,Z 210.368,A -85,B 0,C 180,E1 -7244.105,E2 -7244.105} C_VEL
LIN {X 0,Y 474.587,Z 210.366,A -85,B 0,C 180,E1 -7247.062,E2 -7247.062} C_VEL
LIN {X 0,Y 474.619,Z 210.363,A -85,B 0,C 180,E1 -7249.341,E2 -7249.341} C_VEL
LIN {X 0,Y 474.59,Z 210.368,A -85,B 0,C 180,E1 -7252.615,E2 -7252.615} C_VEL
LIN {X 0,Y 474.636,Z 210.365,A -85,B 0,C 180,E1 -7255.758,E2 -7255.758} C_VEL
LIN {X 0,Y 474.603,Z 210.371,A -85,B 0,C 180,E1 -7258.782,E2 -7258.782} C_VEL
LIN {X 0,Y 474.623,Z 210.372,A -85,B 0,C 180,E1 -7261.715,E2 -7261.715} C_VEL
LIN {X 0,Y 474.679,Z 210.46,A -85,B 0,C 180,E1 -7263.273,E2 -7263.273} C_VEL
LIN {X 0,Y 476.875,Z 221.028,A -85,B 0,C 180,E1 -7265.396,E2 -7265.396} C_VEL
LIN {X 0,Y 477.062,Z 225.679,A -85,B 0,C 180,E1 -7266.254,E2 -7266.254} C_VEL
LIN {X 0,Y 476.23,Z 241.582,A -85,B 0,C 180,E1 -7269.03,E2 -7269.03} C_VEL
LIN {X 0,Y 475.422,Z 261.236,A -85,B 0,C 180,E1 -7272.359,E2 -7272.359} C_VEL
LIN {X 0,Y 475.267,Z 265.9,A -85,B 0,C 180,E1 -7273.121,E2 -7273.121} C_VEL
LIN {X 0,Y 478.042,Z 285.691,A -85,B 0,C 180,E1 -7273.613,E2 -7273.613} C_VEL
LIN {X 0,Y 476.931,Z 376.058,A -85,B 0,C 180,E1 -7275.219,E2 -7275.219} C_VEL
LIN {X 0,Y 476.542,Z 390.092,A -85,B 0,C 180,E1 -7275.643,E2 -7275.643} C_VEL
LIN {X 0,Y 476.13,Z 402.158,A -85,B 0,C 180,E1 -7276.175,E2 -7276.175} C_VEL
LIN {X 0,Y 475.718,Z 413.994,A -85,B 0,C 180,E1 -7276.87,E2 -7276.87} C_VEL
LIN {X 0,Y 475.296,Z 425.536,A -85,B 0,C 180,E1 -7277.732,E2 -7277.732} C_VEL
LIN {X 0,Y 474.926,Z 435.843,A -85,B 0,C 180,E1 -7278.692,E2 -7278.692} C_VEL
LIN {X 0,Y 474.464,Z 445.203,A -85,B 0,C 180,E1 -7279.76,E2 -7279.76} C_VEL
LIN {X 0,Y 474.194,Z 454.346,A -85,B 0,C 180,E1 -7281.046,E2 -7281.046} C_VEL
LIN {X 0,Y 473.999,Z 461.663,A -85,B 0,C 180,E1 -7282.33,E2 -7282.33} C_VEL
LIN {X 0,Y 473.853,Z 467.346,A -85,B 0,C 180,E1 -7283.575,E2 -7283.575} C_VEL
LIN {X 0,Y 473.827,Z 472.08,A -85,B 0,C 180,E1 -7284.893,E2 -7284.893} C_VEL
LIN {X 0,Y 473.748,Z 474.506,A -85,B 0,C 180,E1 -7285.745,E2 -7285.745} C_VEL
LIN {X 0,Y 473.801,Z 476.488,A -85,B 0,C 180,E1 -7286.598,E2 -7286.598} C_VEL
LIN {X 0,Y 473.762,Z 477.976,A -85,B 0,C 180,E1 -7287.448,E2 -7287.448} C_VEL
LIN {X 0,Y 473.756,Z 479.038,A -85,B 0,C 180,E1 -7288.299,E2 -7288.299} C_VEL
LIN {X 0,Y 473.693,Z 479.693,A -85,B 0,C 180,E1 -7289.149,E2 -7289.149} C_VEL
LIN {X 0,Y 473.678,Z 479.933,A -85,B 0,C 180,E1 -7289.999,E2 -7289.999} C_VEL
LIN {X 0,Y 473.693,Z 479.719,A -85,B 0,C 180,E1 -7290.849,E2 -7290.849} C_VEL
LIN {X 0,Y 473.756,Z 479.1,A -85,B 0,C 180,E1 -7291.699,E2 -7291.699} C_VEL
LIN {X 0,Y 473.761,Z 478.073,A -85,B 0,C 180,E1 -7292.55,E2 -7292.55} C_VEL
LIN {X 0,Y 473.819,Z 476.606,A -85,B 0,C 180,E1 -7293.4,E2 -7293.4} C_VEL
LIN {X 0,Y 473.76,Z 473.55,A -85,B 0,C 180,E1 -7294.679,E2 -7294.679} C_VEL
LIN {X 0,Y 473.814,Z 469.402,A -85,B 0,C 180,E1 -7295.959,E2 -7295.959} C_VEL
LIN {X 0,Y 473.998,Z 463.014,A -85,B 0,C 180,E1 -7297.453,E2 -7297.453} C_VEL
LIN {X 0,Y 474.159,Z 456.04,A -85,B 0,C 180,E1 -7298.738,E2 -7298.738} C_VEL
LIN {X 0,Y 474.378,Z 448.911,A -85,B 0,C 180,E1 -7299.809,E2 -7299.809} C_VEL
LIN {X 0,Y 474.732,Z 440.314,A -85,B 0,C 180,E1 -7300.879,E2 -7300.879} C_VEL
LIN {X 0,Y 475.129,Z 429.678,A -85,B 0,C 180,E1 -7301.951,E2 -7301.951} C_VEL
LIN {X 0,Y 475.528,Z 419.162,A -85,B 0,C 180,E1 -7302.807,E2 -7302.807} C_VEL
LIN {X 0,Y 475.96,Z 407.646,A -85,B 0,C 180,E1 -7303.556,E2 -7303.556} C_VEL
LIN {X 0,Y 476.401,Z 394.513,A -85,B 0,C 180,E1 -7304.196,E2 -7304.196} C_VEL
LIN {X 0,Y 476.791,Z 381.427,A -85,B 0,C 180,E1 -7304.647,E2 -7304.647} C_VEL
LIN {X 0,Y 477.031,Z 367.371,A -85,B 0,C 180,E1 -7304.94,E2 -7304.94} C_VEL
LIN {X 0,Y 477.74,Z 284.803,A -85,B 0,C 180,E1 -7306.33,E2 -7306.33} C_VEL
LIN {X 0,Y 475.277,Z 267.441,A -85,B 0,C 180,E1 -7306.734,E2 -7306.734} C_VEL
LIN {X 0,Y 475.923,Z 250.083,A -85,B 0,C 180,E1 -7309.607,E2 -7309.607} C_VEL
LIN {X 0,Y 476.735,Z 231.284,A -85,B 0,C 180,E1 -7312.765,E2 -7312.765} C_VEL
LIN {X 0,Y 477.072,Z 223.837,A -85,B 0,C 180,E1 -7314.027,E2 -7314.027} C_VEL
LIN {X 0,Y 476.201,Z 217.826,A -85,B 0,C 180,E1 -7315.106,E2 -7315.106} C_VEL
LIN {X 0,Y 474.688,Z 210.359,A -85,B 0,C 180,E1 -7316.487,E2 -7316.487} C_VEL
LIN {X 0,Y 474.617,Z 210.364,A -85,B 0,C 180,E1 -7319.251,E2 -7319.251} C_VEL
LIN {X 0,Y 474.612,Z 210.354,A -85,B 0,C 180,E1 -7322.43,E2 -7322.43} C_VEL
LIN {X 0,Y 474.607,Z 210.359,A -85,B 0,C 180,E1 -7325.468,E2 -7325.468} C_VEL
LIN {X 0,Y 474.603,Z 210.36,A -85,B 0,C 180,E1 -7328.457,E2 -7328.457} C_VEL
LIN {X 0,Y 474.603,Z 210.366,A -85,B 0,C 180,E1 -7331.786,E2 -7331.786} C_VEL
LIN {X 0,Y 474.61,Z 210.361,A -85,B 0,C 180,E1 -7334.701,E2 -7334.701} C_VEL
LIN {X 0,Y 474.581,Z 210.362,A -85,B 0,C 180,E1 -7337.767,E2 -7337.767} C_VEL
LIN {X 0,Y 474.614,Z 210.36,A -85,B 0,C 180,E1 -7340.451,E2 -7340.451} C_VEL
LIN {X 0,Y 474.581,Z 210.358,A -85,B 0,C 180,E1 -7343.676,E2 -7343.676} C_VEL
LIN {X 0,Y 474.616,Z 210.361,A -85,B 0,C 180,E1 -7346.778,E2 -7346.778} C_VEL
LIN {X 0,Y 474.586,Z 210.356,A -85,B 0,C 180,E1 -7349.768,E2 -7349.768} C_VEL
LIN {X 0,Y 474.593,Z 210.36,A -85,B 0,C 180,E1 -7352.684,E2 -7352.684} C_VEL
LIN {X 0,Y 474.616,Z 210.358,A -85,B 0,C 180,E1 -7355.505,E2 -7355.505} C_VEL
LIN {X 0,Y 474.624,Z 210.352,A -85,B 0,C 180,E1 -7358.884,E2 -7358.884} C_VEL
LIN {X 0,Y 474.63,Z 210.358,A -85,B 0,C 180,E1 -7361.883,E2 -7361.883} C_VEL
LIN {X 0,Y 474.686,Z 210.351,A -85,B 0,C 180,E1 -7364.544,E2 -7364.544} C_VEL
LIN {X 0,Y 474.694,Z 210.346,A -85,B 0,C 180,E1 -7368.037,E2 -7368.037} C_VEL
LIN {X 0,Y 474.697,Z 210.35,A -85,B 0,C 180,E1 -7371.486,E2 -7371.486} C_VEL
LIN {X 0,Y 474.719,Z 210.342,A -85,B 0,C 180,E1 -7374.052,E2 -7374.052} C_VEL
LIN {X 0,Y 474.872,Z 210.326,A -85,B 0,C 180,E1 -7377.455,E2 -7377.455} C_VEL
LIN {X 0,Y 474.87,Z 210.332,A -85,B 0,C 180,E1 -7380,E2 -7380} C_VEL
LIN {X 0,Y 474.871,Z 210.318,A -85,B 0,C 180,E1 -7382.545,E2 -7382.545} C_VEL
LIN {X 0,Y 474.761,Z 210.344,A -85,B 0,C 180,E1 -7385.948,E2 -7385.948} C_VEL
LIN {X 0,Y 474.717,Z 210.343,A -85,B 0,C 180,E1 -7388.514,E2 -7388.514} C_VEL
LIN {X 0,Y 474.696,Z 210.349,A -85,B 0,C 180,E1 -7391.963,E2 -7391.963} C_VEL
LIN {X 0,Y 474.692,Z 210.353,A -85,B 0,C 180,E1 -7395.456,E2 -7395.456} C_VEL
LIN {X 0,Y 474.655,Z 210.352,A -85,B 0,C 180,E1 -7399.011,E2 -7399.011} C_VEL
LIN {X 0,Y 474.582,Z 210.369,A -85,B 0,C 180,E1 -7401.73,E2 -7401.73} C_VEL
LIN {X 0,Y 474.652,Z 210.352,A -85,B 0,C 180,E1 -7404.494,E2 -7404.494} C_VEL
LIN {X 0,Y 474.674,Z 210.36,A -85,B 0,C 180,E1 -7407.335,E2 -7407.335} C_VEL
LIN {X 0,Y 474.598,Z 210.363,A -85,B 0,C 180,E1 -7410.811,E2 -7410.811} C_VEL
LIN {X 0,Y 474.633,Z 210.356,A -85,B 0,C 180,E1 -7413.985,E2 -7413.985} C_VEL
LIN {X 0,Y 474.57,Z 210.373,A -85,B 0,C 180,E1 -7416.901,E2 -7416.901} C_VEL
LIN {X 0,Y 474.623,Z 210.364,A -85,B 0,C 180,E1 -7419.649,E2 -7419.649} C_VEL
LIN {X 0,Y 474.628,Z 210.364,A -85,B 0,C 180,E1 -7422.933,E2 -7422.933} C_VEL
LIN {X 0,Y 474.611,Z 210.363,A -85,B 0,C 180,E1 -7425.897,E2 -7425.897} C_VEL
LIN {X 0,Y 474.626,Z 210.364,A -85,B 0,C 180,E1 -7429.042,E2 -7429.042} C_VEL
LIN {X 0,Y 474.608,Z 210.362,A -85,B 0,C 180,E1 -7431.705,E2 -7431.705} C_VEL
LIN {X 0,Y 474.624,Z 210.366,A -85,B 0,C 180,E1 -7434.727,E2 -7434.727} C_VEL
LIN {X 0,Y 474.748,Z 210.392,A -85,B 0,C 180,E1 -7437.798,E2 -7437.798} C_VEL
LIN {X 0,Y 475.196,Z 221.931,A -85,B 0,C 180,E1 -7439.168,E2 -7439.168} C_VEL
LIN {X 0,Y 478.34,Z 239.762,A -85,B 0,C 180,E1 -7439.586,E2 -7439.586} C_VEL
LIN {X 0,Y 477.728,Z 308.09,A -85,B 0,C 180,E1 -7440.62,E2 -7440.62} C_VEL
LIN {X 0,Y 477.005,Z 313.944,A -85,B 0,C 180,E1 -7440.681,E2 -7440.681} C_VEL
LIN {X 0,Y 471.313,Z 332.922,A -85,B 0,C 180,E1 -7440.791,E2 -7440.791} C_VEL
LIN {X 0,Y 470.63,Z 338.689,A -85,B 0,C 180,E1 -7440.912,E2 -7440.912} C_VEL
LIN {X 0,Y 470.347,Z 350.623,A -85,B 0,C 180,E1 -7441.315,E2 -7441.315} C_VEL
LIN {X 0,Y 469.999,Z 363.1,A -85,B 0,C 180,E1 -7441.915,E2 -7441.915} C_VEL
LIN {X 0,Y 469.547,Z 375.518,A -85,B 0,C 180,E1 -7442.718,E2 -7442.718} C_VEL
LIN {X 0,Y 468.995,Z 385.435,A -85,B 0,C 180,E1 -7443.526,E2 -7443.526} C_VEL
LIN {X 0,Y 468.514,Z 395.736,A -85,B 0,C 180,E1 -7444.572,E2 -7444.572} C_VEL
LIN {X 0,Y 467.992,Z 405.774,A -85,B 0,C 180,E1 -7445.845,E2 -7445.845} C_VEL
LIN {X 0,Y 467.661,Z 413.14,A -85,B 0,C 180,E1 -7447.001,E2 -7447.001} C_VEL
LIN {X 0,Y 467.295,Z 420.215,A -85,B 0,C 180,E1 -7448.38,E2 -7448.38} C_VEL
LIN {X 0,Y 467.009,Z 425.781,A -85,B 0,C 180,E1 -7449.751,E2 -7449.751} C_VEL
LIN {X 0,Y 466.853,Z 430.171,A -85,B 0,C 180,E1 -7451.162,E2 -7451.162} C_VEL
LIN {X 0,Y 466.719,Z 433.151,A -85,B 0,C 180,E1 -7452.473,E2 -7452.473} C_VEL
LIN {X 0,Y 466.63,Z 434.64,A -85,B 0,C 180,E1 -7453.373,E2 -7453.373} C_VEL
LIN {X 0,Y 466.619,Z 435.924,A -85,B 0,C 180,E1 -7454.568,E2 -7454.568} C_VEL
LIN {X 0,Y 466.565,Z 436.469,A -85,B 0,C 180,E1 -7456.055,E2 -7456.055} C_VEL
LIN {X 0,Y 466.58,Z 436.212,A -85,B 0,C 180,E1 -7456.943,E2 -7456.943} C_VEL
LIN {X 0,Y 466.678,Z 435.163,A -85,B 0,C 180,E1 -7458.205,E2 -7458.205} C_VEL
LIN {X 0,Y 466.71,Z 433.012,A -85,B 0,C 180,E1 -7459.59,E2 -7459.59} C_VEL
LIN {X 0,Y 466.84,Z 429.958,A -85,B 0,C 180,E1 -7460.906,E2 -7460.906} C_VEL
LIN {X 0,Y 466.989,Z 425.851,A -85,B 0,C 180,E1 -7462.217,E2 -7462.217} C_VEL
LIN {X 0,Y 467.257,Z 419.806,A -85,B 0,C 180,E1 -7463.694,E2 -7463.694} C_VEL
LIN {X 0,Y 467.54,Z 412.76,A -85,B 0,C 180,E1 -7465.043,E2 -7465.043} C_VEL
LIN {X 0,Y 467.916,Z 404.225,A -85,B 0,C 180,E1 -7466.341,E2 -7466.341} C_VEL
LIN {X 0,Y 468.365,Z 395.499,A -85,B 0,C 180,E1 -7467.421,E2 -7467.421} C_VEL
LIN {X 0,Y 468.774,Z 385.963,A -85,B 0,C 180,E1 -7468.39,E2 -7468.39} C_VEL
LIN {X 0,Y 469.289,Z 375.427,A -85,B 0,C 180,E1 -7469.25,E2 -7469.25} C_VEL
LIN {X 0,Y 469.734,Z 363.81,A -85,B 0,C 180,E1 -7470.001,E2 -7470.001} C_VEL
LIN {X 0,Y 470.105,Z 351.874,A -85,B 0,C 180,E1 -7470.59,E2 -7470.59} C_VEL
LIN {X 0,Y 470.374,Z 339.625,A -85,B 0,C 180,E1 -7471.018,E2 -7471.018} C_VEL
LIN {X 0,Y 470.527,Z 326.032,A -85,B 0,C 180,E1 -7471.311,E2 -7471.311} C_VEL
LIN {X 0,Y 471.151,Z 239.314,A -85,B 0,C 180,E1 -7472.637,E2 -7472.637} C_VEL
LIN {X 0,Y 468.032,Z 222.167,A -85,B 0,C 180,E1 -7473.016,E2 -7473.016} C_VEL
LIN {X 0,Y 467.604,Z 211.369,A -85,B 0,C 180,E1 -7474.311,E2 -7474.311} C_VEL
LIN {X 0,Y 467.73,Z 211.222,A -85,B 0,C 180,E1 -7476.038,E2 -7476.038} C_VEL
LIN {X 0,Y 467.674,Z 211.229,A -85,B 0,C 180,E1 -7478.644,E2 -7478.644} C_VEL
LIN {X 0,Y 467.663,Z 211.23,A -85,B 0,C 180,E1 -7482.146,E2 -7482.146} C_VEL
LIN {X 0,Y 467.656,Z 211.231,A -85,B 0,C 180,E1 -7485.885,E2 -7485.885} C_VEL
LIN {X 0,Y 467.628,Z 211.236,A -85,B 0,C 180,E1 -7489.308,E2 -7489.308} C_VEL
LIN {X 0,Y 467.538,Z 211.245,A -85,B 0,C 180,E1 -7492.075,E2 -7492.075} C_VEL
LIN {X 0,Y 467.561,Z 211.244,A -85,B 0,C 180,E1 -7494.891,E2 -7494.891} C_VEL
LIN {X 0,Y 467.552,Z 211.243,A -85,B 0,C 180,E1 -7497.774,E2 -7497.774} C_VEL
LIN {X 0,Y 467.554,Z 211.245,A -85,B 0,C 180,E1 -7501.041,E2 -7501.041} C_VEL
LIN {X 0,Y 467.582,Z 211.243,A -85,B 0,C 180,E1 -7504.24,E2 -7504.24} C_VEL
LIN {X 0,Y 467.527,Z 211.248,A -85,B 0,C 180,E1 -7507.182,E2 -7507.182} C_VEL
LIN {X 0,Y 467.543,Z 211.247,A -85,B 0,C 180,E1 -7510.269,E2 -7510.269} C_VEL
LIN {X 0,Y 467.522,Z 211.249,A -85,B 0,C 180,E1 -7512.569,E2 -7512.569} C_VEL
LIN {X 0,Y 467.568,Z 211.242,A -85,B 0,C 180,E1 -7515.052,E2 -7515.052} C_VEL
LIN {X 0,Y 467.555,Z 211.245,A -85,B 0,C 180,E1 -7518.728,E2 -7518.728} C_VEL
LIN {X 0,Y 467.537,Z 211.248,A -85,B 0,C 180,E1 -7521.952,E2 -7521.952} C_VEL
LIN {X 0,Y 467.529,Z 211.247,A -85,B 0,C 180,E1 -7525.164,E2 -7525.164} C_VEL
LIN {X 0,Y 467.552,Z 211.246,A -85,B 0,C 180,E1 -7528.257,E2 -7528.257} C_VEL
LIN {X 0,Y 467.532,Z 211.247,A -85,B 0,C 180,E1 -7531.247,E2 -7531.247} C_VEL
LIN {X 0,Y 467.567,Z 211.243,A -85,B 0,C 180,E1 -7534.405,E2 -7534.405} C_VEL
LIN {X 0,Y 467.578,Z 211.241,A -85,B 0,C 180,E1 -7536.996,E2 -7536.996} C_VEL
LIN {X 0,Y 467.588,Z 211.307,A -85,B 0,C 180,E1 -7538.798,E2 -7538.798} C_VEL
LIN {X 0,Y 468.574,Z 217.692,A -85,B 0,C 180,E1 -7540.277,E2 -7540.277} C_VEL
LIN {X 0,Y 468.388,Z 226.189,A -85,B 0,C 180,E1 -7542.155,E2 -7542.155} C_VEL
LIN {X 0,Y 471.16,Z 240.524,A -85,B 0,C 180,E1 -7542.506,E2 -7542.506} C_VEL
LIN {X 0,Y 470.037,Z 334.007,A -85,B 0,C 180,E1 -7544.136,E2 -7544.136} C_VEL
LIN {X 0,Y 469.807,Z 347.32,A -85,B 0,C 180,E1 -7544.546,E2 -7544.546} C_VEL
LIN {X 0,Y 469.499,Z 359.573,A -85,B 0,C 180,E1 -7545.091,E2 -7545.091} C_VEL
LIN {X 0,Y 469.103,Z 371.428,A -85,B 0,C 180,E1 -7545.799,E2 -7545.799} C_VEL
LIN {X 0,Y 468.646,Z 382.88,A -85,B 0,C 180,E1 -7546.669,E2 -7546.669} C_VEL
LIN {X 0,Y 468.304,Z 392.869,A -85,B 0,C 180,E1 -7547.615,E2 -7547.615} C_VEL
LIN {X 0,Y 467.905,Z 402.479,A -85,B 0,C 180,E1 -7548.74,E2 -7548.74} C_VEL
LIN {X 0,Y 467.528,Z 411.511,A -85,B 0,C 180,E1 -7550.045,E2 -7550.045} C_VEL
LIN {X 0,Y 467.247,Z 418.726,A -85,B 0,C 180,E1 -7551.349,E2 -7551.349} C_VEL
LIN {X 0,Y 467.026,Z 424.466,A -85,B 0,C 180,E1 -7552.651,E2 -7552.651} C_VEL
LIN {X 0,Y 466.936,Z 428.967,A -85,B 0,C 180,E1 -7553.952,E2 -7553.952} C_VEL
LIN {X 0,Y 466.793,Z 431.347,A -85,B 0,C 180,E1 -7554.817,E2 -7554.817} C_VEL
LIN {X 0,Y 466.765,Z 433.283,A -85,B 0,C 180,E1 -7555.682,E2 -7555.682} C_VEL
LIN {X 0,Y 466.799,Z 434.732,A -85,B 0,C 180,E1 -7556.547,E2 -7556.547} C_VEL
LIN {X 0,Y 466.738,Z 435.772,A -85,B 0,C 180,E1 -7557.411,E2 -7557.411} C_VEL
LIN {X 0,Y 466.7,Z 436.414,A -85,B 0,C 180,E1 -7558.274,E2 -7558.274} C_VEL
LIN {X 0,Y 466.631,Z 436.637,A -85,B 0,C 180,E1 -7559.137,E2 -7559.137} C_VEL
LIN {X 0,Y 466.614,Z 436.415,A -85,B 0,C 180,E1 -7560,E2 -7560} C_VEL
LIN {X 0,Y 466.636,Z 435.795,A -85,B 0,C 180,E1 -7560.863,E2 -7560.863} C_VEL
LIN {X 0,Y 466.71,Z 434.774,A -85,B 0,C 180,E1 -7561.726,E2 -7561.726} C_VEL
LIN {X 0,Y 466.856,Z 433.293,A -85,B 0,C 180,E1 -7562.588,E2 -7562.588} C_VEL
LIN {X 0,Y 466.939,Z 430.262,A -85,B 0,C 180,E1 -7563.883,E2 -7563.883} C_VEL
LIN {X 0,Y 467.047,Z 426.15,A -85,B 0,C 180,E1 -7565.18,E2 -7565.18} C_VEL
LIN {X 0,Y 467.323,Z 420.833,A -85,B 0,C 180,E1 -7566.476,E2 -7566.476} C_VEL
LIN {X 0,Y 467.504,Z 414.15,A -85,B 0,C 180,E1 -7567.776,E2 -7567.776} C_VEL
LIN {X 0,Y 467.895,Z 405.821,A -85,B 0,C 180,E1 -7569.074,E2 -7569.074} C_VEL
LIN {X 0,Y 468.261,Z 397.242,A -85,B 0,C 180,E1 -7570.157,E2 -7570.157} C_VEL
LIN {X 0,Y 468.68,Z 386.661,A -85,B 0,C 180,E1 -7571.241,E2 -7571.241} C_VEL
LIN {X 0,Y 469.174,Z 376.162,A -85,B 0,C 180,E1 -7572.105,E2 -7572.105} C_VEL
LIN {X 0,Y 469.542,Z 364.543,A -85,B 0,C 180,E1 -7572.864,E2 -7572.864} C_VEL
LIN {X 0,Y 469.975,Z 351.363,A -85,B 0,C 180,E1 -7573.511,E2 -7573.511} C_VEL
LIN {X 0,Y 470.159,Z 338.976,A -85,B 0,C 180,E1 -7573.948,E2 -7573.948} C_VEL
LIN {X 0,Y 470.381,Z 323.685,A -85,B 0,C 180,E1 -7574.272,E2 -7574.272} C_VEL
LIN {X 0,Y 471.722,Z 241.289,A -85,B 0,C 180,E1 -7575.785,E2 -7575.785} C_VEL
LIN {X 0,Y 468.957,Z 228.43,A -85,B 0,C 180,E1 -7576.196,E2 -7576.196} C_VEL
LIN {X 0,Y 469.273,Z 221.34,A -85,B 0,C 180,E1 -7577.879,E2 -7577.879} C_VEL
LIN {X 0,Y 468.602,Z 215.9,A -85,B 0,C 180,E1 -7579.266,E2 -7579.266} C_VEL
LIN {X 0,Y 467.652,Z 211.237,A -85,B 0,C 180,E1 -7580.566,E2 -7580.566} C_VEL
LIN {X 0,Y 467.567,Z 211.246,A -85,B 0,C 180,E1 -7583.944,E2 -7583.944} C_VEL
LIN {X 0,Y 467.619,Z 211.239,A -85,B 0,C 180,E1 -7586.8,E2 -7586.8} C_VEL
LIN {X 0,Y 467.559,Z 211.245,A -85,B 0,C 180,E1 -7589.738,E2 -7589.738} C_VEL
LIN {X 0,Y 467.589,Z 211.241,A -85,B 0,C 180,E1 -7592.758,E2 -7592.758} C_VEL
LIN {X 0,Y 467.559,Z 211.246,A -85,B 0,C 180,E1 -7595.889,E2 -7595.889} C_VEL
LIN {X 0,Y 467.587,Z 211.237,A -85,B 0,C 180,E1 -7599.144,E2 -7599.144} C_VEL
LIN {X 0,Y 467.592,Z 211.241,A -85,B 0,C 180,E1 -7602.566,E2 -7602.566} C_VEL
LIN {X 0,Y 467.57,Z 211.24,A -85,B 0,C 180,E1 -7605.052,E2 -7605.052} C_VEL
LIN {X 0,Y 467.578,Z 211.242,A -85,B 0,C 180,E1 -7608.596,E2 -7608.596} C_VEL
LIN {X 0,Y 467.567,Z 211.245,A -85,B 0,C 180,E1 -7611.955,E2 -7611.955} C_VEL
LIN {X 0,Y 467.567,Z 211.243,A -85,B 0,C 180,E1 -7615.167,E2 -7615.167} C_VEL
LIN {X 0,Y 467.588,Z 211.247,A -85,B 0,C 180,E1 -7618.259,E2 -7618.259} C_VEL
LIN {X 0,Y 467.56,Z 211.251,A -85,B 0,C 180,E1 -7621.248,E2 -7621.248} C_VEL
LIN {X 0,Y 467.639,Z 211.261,A -85,B 0,C 180,E1 -7622.924,E2 -7622.924} C_VEL
LIN {X 0,Y 470.001,Z 222.488,A -85,B 0,C 180,E1 -7625.247,E2 -7625.247} C_VEL
LIN {X 0,Y 470.293,Z 225.804,A -85,B 0,C 180,E1 -7625.884,E2 -7625.884} C_VEL
LIN {X 0,Y 469.364,Z 241.78,A -85,B 0,C 180,E1 -7628.736,E2 -7628.736} C_VEL
LIN {X 0,Y 468.523,Z 259.848,A -85,B 0,C 180,E1 -7631.864,E2 -7631.864} C_VEL
LIN {X 0,Y 468.308,Z 265.537,A -85,B 0,C 180,E1 -7632.814,E2 -7632.814} C_VEL
LIN {X 0,Y 470.751,Z 282.219,A -85,B 0,C 180,E1 -7633.251,E2 -7633.251} C_VEL
LIN {X 0,Y 471.255,Z 287.336,A -85,B 0,C 180,E1 -7633.371,E2 -7633.371} C_VEL
LIN {X 0,Y 470.075,Z 375.993,A -85,B 0,C 180,E1 -7634.998,E2 -7634.998} C_VEL
LIN {X 0,Y 469.663,Z 389.844,A -85,B 0,C 180,E1 -7635.428,E2 -7635.428} C_VEL
LIN {X 0,Y 469.176,Z 402.821,A -85,B 0,C 180,E1 -7636.021,E2 -7636.021} C_VEL
LIN {X 0,Y 468.7,Z 415.226,A -85,B 0,C 180,E1 -7636.78,E2 -7636.78} C_VEL
LIN {X 0,Y 468.294,Z 425.721,A -85,B 0,C 180,E1 -7637.593,E2 -7637.593} C_VEL
LIN {X 0,Y 467.925,Z 435.474,A -85,B 0,C 180,E1 -7638.52,E2 -7638.52} C_VEL
LIN {X 0,Y 467.432,Z 444.834,A -85,B 0,C 180,E1 -7639.605,E2 -7639.605} C_VEL
LIN {X 0,Y 467.145,Z 453.983,A -85,B 0,C 180,E1 -7640.91,E2 -7640.91} C_VEL
LIN {X 0,Y 466.93,Z 461.305,A -85,B 0,C 180,E1 -7642.214,E2 -7642.214} C_VEL
LIN {X 0,Y 466.778,Z 467.392,A -85,B 0,C 180,E1 -7643.578,E2 -7643.578} C_VEL
LIN {X 0,Y 466.735,Z 471.745,A -85,B 0,C 180,E1 -7644.816,E2 -7644.816} C_VEL
LIN {X 0,Y 466.658,Z 474.176,A -85,B 0,C 180,E1 -7645.681,E2 -7645.681} C_VEL
LIN {X 0,Y 466.697,Z 476.16,A -85,B 0,C 180,E1 -7646.546,E2 -7646.546} C_VEL
LIN {X 0,Y 466.681,Z 477.649,A -85,B 0,C 180,E1 -7647.41,E2 -7647.41} C_VEL
LIN {X 0,Y 466.661,Z 478.712,A -85,B 0,C 180,E1 -7648.273,E2 -7648.273} C_VEL
LIN {X 0,Y 466.624,Z 479.368,A -85,B 0,C 180,E1 -7649.136,E2 -7649.136} C_VEL
LIN {X 0,Y 466.607,Z 479.603,A -85,B 0,C 180,E1 -7649.999,E2 -7649.999} C_VEL
LIN {X 0,Y 466.624,Z 479.383,A -85,B 0,C 180,E1 -7650.862,E2 -7650.862} C_VEL
LIN {X 0,Y 466.661,Z 478.758,A -85,B 0,C 180,E1 -7651.725,E2 -7651.725} C_VEL
LIN {X 0,Y 466.681,Z 477.725,A -85,B 0,C 180,E1 -7652.588,E2 -7652.588} C_VEL
LIN {X 0,Y 466.727,Z 476.24,A -85,B 0,C 180,E1 -7653.452,E2 -7653.452} C_VEL
LIN {X 0,Y 466.687,Z 473.162,A -85,B 0,C 180,E1 -7654.75,E2 -7654.75} C_VEL
LIN {X 0,Y 466.732,Z 468.985,A -85,B 0,C 180,E1 -7656.05,E2 -7656.05} C_VEL
LIN {X 0,Y 466.904,Z 462.558,A -85,B 0,C 180,E1 -7657.567,E2 -7657.567} C_VEL
LIN {X 0,Y 467.093,Z 455.542,A -85,B 0,C 180,E1 -7658.871,E2 -7658.871} C_VEL
LIN {X 0,Y 467.316,Z 448.362,A -85,B 0,C 180,E1 -7659.958,E2 -7659.958} C_VEL
LIN {X 0,Y 467.708,Z 439.683,A -85,B 0,C 180,E1 -7661.044,E2 -7661.044} C_VEL
LIN {X 0,Y 468.139,Z 428.981,A -85,B 0,C 180,E1 -7662.132,E2 -7662.132} C_VEL
LIN {X 0,Y 468.571,Z 418.383,A -85,B 0,C 180,E1 -7663.001,E2 -7663.001} C_VEL
LIN {X 0,Y 469.143,Z 405.06,A -85,B 0,C 180,E1 -7663.867,E2 -7663.867} C_VEL
LIN {X 0,Y 469.528,Z 392.684,A -85,B 0,C 180,E1 -7664.464,E2 -7664.464} C_VEL
LIN {X 0,Y 469.989,Z 379.853,A -85,B 0,C 180,E1 -7664.892,E2 -7664.892} C_VEL
LIN {X 0,Y 470.154,Z 366.436,A -85,B 0,C 180,E1 -7665.164,E2 -7665.164} C_VEL
LIN {X 0,Y 470.947,Z 286.474,A -85,B 0,C 180,E1 -7666.517,E2 -7666.517} C_VEL
LIN {X 0,Y 468.306,Z 267.332,A -85,B 0,C 180,E1 -7666.948,E2 -7666.948} C_VEL
LIN {X 0,Y 469.022,Z 248.252,A -85,B 0,C 180,E1 -7670.159,E2 -7670.159} C_VEL
LIN {X 0,Y 469.925,Z 229.551,A -85,B 0,C 180,E1 -7673.347,E2 -7673.347} C_VEL
LIN {X 0,Y 470.039,Z 223.36,A -85,B 0,C 180,E1 -7674.423,E2 -7674.423} C_VEL
LIN {X 0,Y 467.659,Z 211.233,A -85,B 0,C 180,E1 -7676.706,E2 -7676.706} C_VEL
LIN {X 0,Y 467.55,Z 211.248,A -85,B 0,C 180,E1 -7679.737,E2 -7679.737} C_VEL
LIN {X 0,Y 467.58,Z 211.227,A -85,B 0,C 180,E1 -7682.757,E2 -7682.757} C_VEL
LIN {X 0,Y 467.546,Z 211.244,A -85,B 0,C 180,E1 -7685.889,E2 -7685.889} C_VEL
LIN {X 0,Y 467.547,Z 211.239,A -85,B 0,C 180,E1 -7689.147,E2 -7689.147} C_VEL
LIN {X 0,Y 467.561,Z 211.245,A -85,B 0,C 180,E1 -7691.403,E2 -7691.403} C_VEL
LIN {X 0,Y 467.559,Z 211.24,A -85,B 0,C 180,E1 -7694.947,E2 -7694.947} C_VEL
LIN {X 0,Y 467.557,Z 211.232,A -85,B 0,C 180,E1 -7698.595,E2 -7698.595} C_VEL
LIN {X 0,Y 467.556,Z 211.24,A -85,B 0,C 180,E1 -7701.955,E2 -7701.955} C_VEL
LIN {X 0,Y 467.55,Z 211.237,A -85,B 0,C 180,E1 -7705.166,E2 -7705.166} C_VEL
LIN {X 0,Y 467.571,Z 211.236,A -85,B 0,C 180,E1 -7708.259,E2 -7708.259} C_VEL
LIN {X 0,Y 467.535,Z 211.237,A -85,B 0,C 180,E1 -7711.248,E2 -7711.248} C_VEL
LIN {X 0,Y 467.567,Z 211.238,A -85,B 0,C 180,E1 -7714.401,E2 -7714.401} C_VEL
LIN {X 0,Y 467.562,Z 211.231,A -85,B 0,C 180,E1 -7716.995,E2 -7716.995} C_VEL
LIN {X 0,Y 467.608,Z 211.228,A -85,B 0,C 180,E1 -7719.777,E2 -7719.777} C_VEL
LIN {X 0,Y 467.577,Z 211.241,A -85,B 0,C 180,E1 -7722.506,E2 -7722.506} C_VEL
LIN {X 0,Y 467.582,Z 211.226,A -85,B 0,C 180,E1 -7725.196,E2 -7725.196} C_VEL
LIN {X 0,Y 467.646,Z 211.223,A -85,B 0,C 180,E1 -7727.854,E2 -7727.854} C_VEL
LIN {X 0,Y 467.655,Z 211.227,A -85,B 0,C 180,E1 -7731.357,E2 -7731.357} C_VEL
LIN {X 0,Y 467.684,Z 211.218,A -85,B 0,C 180,E1 -7733.962,E2 -7733.962} C_VEL
LIN {X 0,Y 467.838,Z 211.202,A -85,B 0,C 180,E1 -7737.417,E2 -7737.417} C_VEL
LIN {X 0,Y 467.839,Z 211.208,A -85,B 0,C 180,E1 -7740,E2 -7740} C_VEL
LIN {X 0,Y 467.812,Z 211.197,A -85,B 0,C 180,E1 -7742.583,E2 -7742.583} C_VEL
LIN {X 0,Y 467.726,Z 211.222,A -85,B 0,C 180,E1 -7746.038,E2 -7746.038} C_VEL
LIN {X 0,Y 467.671,Z 211.22,A -85,B 0,C 180,E1 -7748.643,E2 -7748.643} C_VEL
LIN {X 0,Y 467.646,Z 211.229,A -85,B 0,C 180,E1 -7752.358,E2 -7752.358} C_VEL
LIN {X 0,Y 467.641,Z 211.228,A -85,B 0,C 180,E1 -7755.886,E2 -7755.886} C_VEL
LIN {X 0,Y 467.614,Z 211.231,A -85,B 0,C 180,E1 -7759.308,E2 -7759.308} C_VEL
LIN {X 0,Y 467.528,Z 211.243,A -85,B 0,C 180,E1 -7762.075,E2 -7762.075} C_VEL
LIN {X 0,Y 467.597,Z 211.231,A -85,B 0,C 180,E1 -7764.888,E2 -7764.888} C_VEL
LIN {X 0,Y 467.613,Z 211.234,A -85,B 0,C 180,E1 -7767.77,E2 -7767.77} C_VEL
LIN {X 0,Y 467.562,Z 211.242,A -85,B 0,C 180,E1 -7771.046,E2 -7771.046} C_VEL
LIN {X 0,Y 467.584,Z 211.233,A -85,B 0,C 180,E1 -7774.243,E2 -7774.243} C_VEL
LIN {X 0,Y 467.545,Z 211.248,A -85,B 0,C 180,E1 -7777.188,E2 -7777.188} C_VEL
LIN {X 0,Y 467.573,Z 211.241,A -85,B 0,C 180,E1 -7780.266,E2 -7780.266} C_VEL
LIN {X 0,Y 467.583,Z 211.237,A -85,B 0,C 180,E1 -7782.568,E2 -7782.568} C_VEL
LIN {X 0,Y 467.567,Z 211.243,A -85,B 0,C 180,E1 -7785.054,E2 -7785.054} C_VEL
LIN {X 0,Y 467.586,Z 211.238,A -85,B 0,C 180,E1 -7787.441,E2 -7787.441} C_VEL
LIN {X 0,Y 467.58,Z 211.244,A -85,B 0,C 180,E1 -7790.857,E2 -7790.857} C_VEL
LIN {X 0,Y 467.558,Z 211.245,A -85,B 0,C 180,E1 -7794.262,E2 -7794.262} C_VEL
LIN {X 0,Y 467.709,Z 211.308,A -85,B 0,C 180,E1 -7797.636,E2 -7797.636} C_VEL
LIN {X 0,Y 468.144,Z 216.995,A -85,B 0,C 180,E1 -7798.304,E2 -7798.304} C_VEL
LIN {X 0,Y 468.329,Z 222.247,A -85,B 0,C 180,E1 -7798.905,E2 -7798.905} C_VEL
LIN {X 0,Y 471.555,Z 239.853,A -85,B 0,C 180,E1 -7799.319,E2 -7799.319} C_VEL
LIN {X 0,Y 470.742,Z 332.418,A -85,B 0,C 180,E1 -7800.761,E2 -7800.761} C_VEL
LIN {X 0,Y 470.63,Z 338.689,A -85,B 0,C 180,E1 -7800.912,E2 -7800.912} C_VEL
LIN {X 0,Y 469.914,Z 344.434,A -85,B 0,C 180,E1 -7801.061,E2 -7801.061} C_VEL
LIN {X 0,Y 466.956,Z 353.693,A -85,B 0,C 180,E1 -7801.31,E2 -7801.31} C_VEL
LIN {X 0,Y 463.895,Z 362.673,A -85,B 0,C 180,E1 -7801.655,E2 -7801.655} C_VEL
LIN {X 0,Y 463.021,Z 367.974,A -85,B 0,C 180,E1 -7801.953,E2 -7801.953} C_VEL
LIN {X 0,Y 462.461,Z 379.205,A -85,B 0,C 180,E1 -7802.755,E2 -7802.755} C_VEL
LIN {X 0,Y 461.892,Z 389.697,A -85,B 0,C 180,E1 -7803.696,E2 -7803.696} C_VEL
LIN {X 0,Y 461.449,Z 399.277,A -85,B 0,C 180,E1 -7804.759,E2 -7804.759} C_VEL
LIN {X 0,Y 460.906,Z 408.333,A -85,B 0,C 180,E1 -7806.005,E2 -7806.005} C_VEL
LIN {X 0,Y 460.52,Z 416.14,A -85,B 0,C 180,E1 -7807.336,E2 -7807.336} C_VEL
LIN {X 0,Y 460.199,Z 422.465,A -85,B 0,C 180,E1 -7808.682,E2 -7808.682} C_VEL
LIN {X 0,Y 459.929,Z 427.011,A -85,B 0,C 180,E1 -7809.892,E2 -7809.892} C_VEL
LIN {X 0,Y 459.79,Z 431.291,A -85,B 0,C 180,E1 -7811.387,E2 -7811.387} C_VEL
LIN {X 0,Y 459.574,Z 434.663,A -85,B 0,C 180,E1 -7813.11,E2 -7813.11} C_VEL
LIN {X 0,Y 459.524,Z 436.2,A -85,B 0,C 180,E1 -7814.48,E2 -7814.48} C_VEL
LIN {X 0,Y 459.483,Z 436.765,A -85,B 0,C 180,E1 -7815.835,E2 -7815.835} C_VEL
LIN {X 0,Y 459.489,Z 436.634,A -85,B 0,C 180,E1 -7816.738,E2 -7816.738} C_VEL
LIN {X 0,Y 459.591,Z 435.562,A -85,B 0,C 180,E1 -7818.15,E2 -7818.15} C_VEL
LIN {X 0,Y 459.631,Z 433.707,A -85,B 0,C 180,E1 -7819.428,E2 -7819.428} C_VEL
LIN {X 0,Y 459.735,Z 430.803,A -85,B 0,C 180,E1 -7820.764,E2 -7820.764} C_VEL
LIN {X 0,Y 459.897,Z 426.855,A -85,B 0,C 180,E1 -7822.096,E2 -7822.096} C_VEL
LIN {X 0,Y 460.118,Z 421.764,A -85,B 0,C 180,E1 -7823.42,E2 -7823.42} C_VEL
LIN {X 0,Y 460.425,Z 415.344,A -85,B 0,C 180,E1 -7824.746,E2 -7824.746} C_VEL
LIN {X 0,Y 460.765,Z 407.409,A -85,B 0,C 180,E1 -7826.065,E2 -7826.065} C_VEL
LIN {X 0,Y 461.195,Z 399.299,A -85,B 0,C 180,E1 -7827.162,E2 -7827.162} C_VEL
LIN {X 0,Y 461.662,Z 389.362,A -85,B 0,C 180,E1 -7828.256,E2 -7828.256} C_VEL
LIN {X 0,Y 462.248,Z 378.223,A -85,B 0,C 180,E1 -7829.239,E2 -7829.239} C_VEL
LIN {X 0,Y 462.718,Z 367.33,A -85,B 0,C 180,E1 -7830.001,E2 -7830.001} C_VEL
LIN {X 0,Y 463.087,Z 355.163,A -85,B 0,C 180,E1 -7830.653,E2 -7830.653} C_VEL
LIN {X 0,Y 463.432,Z 342.581,A -85,B 0,C 180,E1 -7831.141,E2 -7831.141} C_VEL
LIN {X 0,Y 463.635,Z 329.462,A -85,B 0,C 180,E1 -7831.467,E2 -7831.467} C_VEL
LIN {X 0,Y 464.423,Z 240.902,A -85,B 0,C 180,E1 -7832.839,E2 -7832.839} C_VEL
LIN {X 0,Y 461.059,Z 222.257,A -85,B 0,C 180,E1 -7833.252,E2 -7833.252} C_VEL
LIN {X 0,Y 460.655,Z 212.706,A -85,B 0,C 180,E1 -7834.376,E2 -7834.376} C_VEL
LIN {X 0,Y 460.579,Z 212.115,A -85,B 0,C 180,E1 -7834.486,E2 -7834.486} C_VEL
LIN {X 0,Y 460.653,Z 212.106,A -85,B 0,C 180,E1 -7837.012,E2 -7837.012} C_VEL
LIN {X 0,Y 460.611,Z 212.109,A -85,B 0,C 180,E1 -7839.663,E2 -7839.663} C_VEL
LIN {X 0,Y 460.603,Z 212.109,A -85,B 0,C 180,E1 -7842.436,E2 -7842.436} C_VEL
LIN {X 0,Y 460.608,Z 212.109,A -85,B 0,C 180,E1 -7845.998,E2 -7845.998} C_VEL
LIN {X 0,Y 460.574,Z 212.114,A -85,B 0,C 180,E1 -7849.616,E2 -7849.616} C_VEL
LIN {X 0,Y 460.514,Z 212.122,A -85,B 0,C 180,E1 -7852.429,E2 -7852.429} C_VEL
LIN {X 0,Y 460.539,Z 212.117,A -85,B 0,C 180,E1 -7855.793,E2 -7855.793} C_VEL
LIN {X 0,Y 460.526,Z 212.121,A -85,B 0,C 180,E1 -7859.233,E2 -7859.233} C_VEL
LIN {X 0,Y 460.524,Z 212.122,A -85,B 0,C 180,E1 -7862.286,E2 -7862.286} C_VEL
LIN {X 0,Y 460.51,Z 212.121,A -85,B 0,C 180,E1 -7865.447,E2 -7865.447} C_VEL
LIN {X 0,Y 460.489,Z 212.125,A -85,B 0,C 180,E1 -7868.888,E2 -7868.888} C_VEL
LIN {X 0,Y 460.501,Z 212.122,A -85,B 0,C 180,E1 -7871.597,E2 -7871.597} C_VEL
LIN {X 0,Y 460.512,Z 212.122,A -85,B 0,C 180,E1 -7874.59,E2 -7874.59} C_VEL
LIN {X 0,Y 460.476,Z 212.128,A -85,B 0,C 180,E1 -7877.813,E2 -7877.813} C_VEL
LIN {X 0,Y 460.479,Z 212.126,A -85,B 0,C 180,E1 -7880.132,E2 -7880.132} C_VEL
LIN {X 0,Y 460.479,Z 212.127,A -85,B 0,C 180,E1 -7882.529,E2 -7882.529} C_VEL
LIN {X 0,Y 460.518,Z 212.123,A -85,B 0,C 180,E1 -7885.621,E2 -7885.621} C_VEL
LIN {X 0,Y 460.51,Z 212.121,A -85,B 0,C 180,E1 -7888.742,E2 -7888.742} C_VEL
LIN {X 0,Y 460.502,Z 212.123,A -85,B 0,C 180,E1 -7891.763,E2 -7891.763} C_VEL
LIN {X 0,Y 460.517,Z 212.12,A -85,B 0,C 180,E1 -7894.703,E2 -7894.703} C_VEL
LIN {X 0,Y 460.513,Z 212.125,A -85,B 0,C 180,E1 -7897.571,E2 -7897.571} C_VEL
LIN {X 0,Y 460.566,Z 212.276,A -85,B 0,C 180,E1 -7898.682,E2 -7898.682} C_VEL
LIN {X 0,Y 461.594,Z 218.742,A -85,B 0,C 180,E1 -7900.198,E2 -7900.198} C_VEL
LIN {X 0,Y 461.43,Z 226.485,A -85,B 0,C 180,E1 -7901.919,E2 -7901.919} C_VEL
LIN {X 0,Y 464.319,Z 241.472,A -85,B 0,C 180,E1 -7902.294,E2 -7902.294} C_VEL
LIN {X 0,Y 463.117,Z 334.122,A -85,B 0,C 180,E1 -7903.95,E2 -7903.95} C_VEL
LIN {X 0,Y 462.879,Z 347.462,A -85,B 0,C 180,E1 -7904.365,E2 -7904.365} C_VEL
LIN {X 0,Y 462.549,Z 359.749,A -85,B 0,C 180,E1 -7904.918,E2 -7904.918} C_VEL
LIN {X 0,Y 462.102,Z 372.428,A -85,B 0,C 180,E1 -7905.691,E2 -7905.691} C_VEL
LIN {X 0,Y 461.63,Z 383.763,A -85,B 0,C 180,E1 -7906.575,E2 -7906.575} C_VEL
LIN {X 0,Y 461.302,Z 393.398,A -85,B 0,C 180,E1 -7907.509,E2 -7907.509} C_VEL
LIN {X 0,Y 460.914,Z 402.345,A -85,B 0,C 180,E1 -7908.567,E2 -7908.567} C_VEL
LIN {X 0,Y 460.501,Z 411.464,A -85,B 0,C 180,E1 -7909.891,E2 -7909.891} C_VEL
LIN {X 0,Y 460.194,Z 418.781,A -85,B 0,C 180,E1 -7911.215,E2 -7911.215} C_VEL
LIN {X 0,Y 459.963,Z 424.588,A -85,B 0,C 180,E1 -7912.537,E2 -7912.537} C_VEL
LIN {X 0,Y 459.859,Z 429.144,A -85,B 0,C 180,E1 -7913.858,E2 -7913.858} C_VEL
LIN {X 0,Y 459.739,Z 431.55,A -85,B 0,C 180,E1 -7914.737,E2 -7914.737} C_VEL
LIN {X 0,Y 459.674,Z 433.517,A -85,B 0,C 180,E1 -7915.615,E2 -7915.615} C_VEL
LIN {X 0,Y 459.729,Z 435,A -85,B 0,C 180,E1 -7916.494,E2 -7916.494} C_VEL
LIN {X 0,Y 459.659,Z 436.061,A -85,B 0,C 180,E1 -7917.371,E2 -7917.371} C_VEL
LIN {X 0,Y 459.608,Z 436.723,A -85,B 0,C 180,E1 -7918.247,E2 -7918.247} C_VEL
LIN {X 0,Y 459.564,Z 436.975,A -85,B 0,C 180,E1 -7919.124,E2 -7919.124} C_VEL
LIN {X 0,Y 459.545,Z 436.773,A -85,B 0,C 180,E1 -7920,E2 -7920} C_VEL
LIN {X 0,Y 459.569,Z 436.168,A -85,B 0,C 180,E1 -7920.876,E2 -7920.876} C_VEL
LIN {X 0,Y 459.65,Z 435.162,A -85,B 0,C 180,E1 -7921.752,E2 -7921.752} C_VEL
LIN {X 0,Y 459.801,Z 433.706,A -85,B 0,C 180,E1 -7922.628,E2 -7922.628} C_VEL
LIN {X 0,Y 459.878,Z 430.696,A -85,B 0,C 180,E1 -7923.943,E2 -7923.943} C_VEL
LIN {X 0,Y 459.978,Z 426.605,A -85,B 0,C 180,E1 -7925.26,E2 -7925.26} C_VEL
LIN {X 0,Y 460.32,Z 420.417,A -85,B 0,C 180,E1 -7926.77,E2 -7926.77} C_VEL
LIN {X 0,Y 460.556,Z 413.419,A -85,B 0,C 180,E1 -7928.114,E2 -7928.114} C_VEL
LIN {X 0,Y 461.041,Z 404.759,A -85,B 0,C 180,E1 -7929.431,E2 -7929.431} C_VEL
LIN {X 0,Y 461.446,Z 395.866,A -85,B 0,C 180,E1 -7930.531,E2 -7930.531} C_VEL
LIN {X 0,Y 461.933,Z 386.113,A -85,B 0,C 180,E1 -7931.519,E2 -7931.519} C_VEL
LIN {X 0,Y 462.279,Z 376.868,A -85,B 0,C 180,E1 -7932.289,E2 -7932.289} C_VEL
LIN {X 0,Y 462.672,Z 365.404,A -85,B 0,C 180,E1 -7933.059,E2 -7933.059} C_VEL
LIN {X 0,Y 463.132,Z 352.035,A -85,B 0,C 180,E1 -7933.731,E2 -7933.731} C_VEL
LIN {X 0,Y 463.342,Z 339.459,A -85,B 0,C 180,E1 -7934.185,E2 -7934.185} C_VEL
LIN {X 0,Y 463.638,Z 322.927,A -85,B 0,C 180,E1 -7934.54,E2 -7934.54} C_VEL
LIN {X 0,Y 465.036,Z 242.783,A -85,B 0,C 180,E1 -7936.061,E2 -7936.061} C_VEL
LIN {X 0,Y 462.836,Z 231.981,A -85,B 0,C 180,E1 -7936.394,E2 -7936.394} C_VEL
LIN {X 0,Y 462.116,Z 228.917,A -85,B 0,C 180,E1 -7936.517,E2 -7936.517} C_VEL
LIN {X 0,Y 462.366,Z 222.178,A -85,B 0,C 180,E1 -7938.156,E2 -7938.156} C_VEL
LIN {X 0,Y 461.229,Z 215.049,A -85,B 0,C 180,E1 -7940.05,E2 -7940.05} C_VEL
LIN {X 0,Y 460.577,Z 212.118,A -85,B 0,C 180,E1 -7940.896,E2 -7940.896} C_VEL
LIN {X 0,Y 460.536,Z 212.123,A -85,B 0,C 180,E1 -7944.333,E2 -7944.333} C_VEL
LIN {X 0,Y 460.577,Z 212.114,A -85,B 0,C 180,E1 -7947.243,E2 -7947.243} C_VEL
LIN {X 0,Y 460.515,Z 212.124,A -85,B 0,C 180,E1 -7950.24,E2 -7950.24} C_VEL
LIN {X 0,Y 460.534,Z 212.117,A -85,B 0,C 180,E1 -7953.324,E2 -7953.324} C_VEL
LIN {X 0,Y 460.481,Z 212.127,A -85,B 0,C 180,E1 -7956.529,E2 -7956.529} C_VEL
LIN {X 0,Y 460.537,Z 212.119,A -85,B 0,C 180,E1 -7959.862,E2 -7959.862} C_VEL
LIN {X 0,Y 460.517,Z 212.12,A -85,B 0,C 180,E1 -7962.9,E2 -7962.9} C_VEL
LIN {X 0,Y 460.51,Z 212.123,A -85,B 0,C 180,E1 -7965.831,E2 -7965.831} C_VEL
LIN {X 0,Y 460.532,Z 212.118,A -85,B 0,C 180,E1 -7968.988,E2 -7968.988} C_VEL
LIN {X 0,Y 460.521,Z 212.119,A -85,B 0,C 180,E1 -7971.265,E2 -7971.265} C_VEL
LIN {X 0,Y 460.513,Z 212.123,A -85,B 0,C 180,E1 -7974.554,E2 -7974.554} C_VEL
LIN {X 0,Y 460.536,Z 212.124,A -85,B 0,C 180,E1 -7977.715,E2 -7977.715} C_VEL
LIN {X 0,Y 460.531,Z 212.126,A -85,B 0,C 180,E1 -7980.767,E2 -7980.767} C_VEL
LIN {X 0,Y 460.606,Z 212.315,A -85,B 0,C 180,E1 -7982.595,E2 -7982.595} C_VEL
LIN {X 0,Y 462.889,Z 222.757,A -85,B 0,C 180,E1 -7984.841,E2 -7984.841} C_VEL
LIN {X 0,Y 463.433,Z 227.725,A -85,B 0,C 180,E1 -7985.828,E2 -7985.828} C_VEL
LIN {X 0,Y 462.37,Z 244.249,A -85,B 0,C 180,E1 -7988.838,E2 -7988.838} C_VEL
LIN {X 0,Y 461.473,Z 262.399,A -85,B 0,C 180,E1 -7992.036,E2 -7992.036} C_VEL
LIN {X 0,Y 461.379,Z 264.94,A -85,B 0,C 180,E1 -7992.476,E2 -7992.476} C_VEL
LIN {X 0,Y 463.933,Z 281.747,A -85,B 0,C 180,E1 -7992.946,E2 -7992.946} C_VEL
LIN {X 0,Y 464.512,Z 288.404,A -85,B 0,C 180,E1 -7993.106,E2 -7993.106} C_VEL
LIN {X 0,Y 463.232,Z 376.174,A -85,B 0,C 180,E1 -7994.771,E2 -7994.771} C_VEL
LIN {X 0,Y 462.802,Z 389.763,A -85,B 0,C 180,E1 -7995.207,E2 -7995.207} C_VEL
LIN {X 0,Y 462.283,Z 402.597,A -85,B 0,C 180,E1 -7995.809,E2 -7995.809} C_VEL
LIN {X 0,Y 461.773,Z 414.943,A -85,B 0,C 180,E1 -7996.578,E2 -7996.578} C_VEL
LIN {X 0,Y 461.293,Z 425.951,A -85,B 0,C 180,E1 -7997.449,E2 -7997.449} C_VEL
LIN {X 0,Y 460.88,Z 436.157,A -85,B 0,C 180,E1 -7998.454,E2 -7998.454} C_VEL
LIN {X 0,Y 460.342,Z 446.19,A -85,B 0,C 180,E1 -7999.665,E2 -7999.665} C_VEL
LIN {X 0,Y 460.102,Z 453.652,A -85,B 0,C 180,E1 -8000.77,E2 -8000.77} C_VEL
LIN {X 0,Y 459.867,Z 460.98,A -85,B 0,C 180,E1 -8002.093,E2 -8002.093} C_VEL
LIN {X 0,Y 459.675,Z 467.586,A -85,B 0,C 180,E1 -8003.612,E2 -8003.612} C_VEL
LIN {X 0,Y 459.617,Z 472.726,A -85,B 0,C 180,E1 -8005.175,E2 -8005.175} C_VEL
LIN {X 0,Y 459.594,Z 475.84,A -85,B 0,C 180,E1 -8006.492,E2 -8006.492} C_VEL
LIN {X 0,Y 459.601,Z 477.327,A -85,B 0,C 180,E1 -8007.37,E2 -8007.37} C_VEL
LIN {X 0,Y 459.57,Z 478.39,A -85,B 0,C 180,E1 -8008.246,E2 -8008.246} C_VEL
LIN {X 0,Y 459.557,Z 479.045,A -85,B 0,C 180,E1 -8009.123,E2 -8009.123} C_VEL
LIN {X 0,Y 459.538,Z 479.269,A -85,B 0,C 180,E1 -8009.999,E2 -8009.999} C_VEL
LIN {X 0,Y 459.556,Z 479.042,A -85,B 0,C 180,E1 -8010.875,E2 -8010.875} C_VEL
LIN {X 0,Y 459.57,Z 478.407,A -85,B 0,C 180,E1 -8011.752,E2 -8011.752} C_VEL
LIN {X 0,Y 459.603,Z 477.364,A -85,B 0,C 180,E1 -8012.628,E2 -8012.628} C_VEL
LIN {X 0,Y 459.623,Z 475.855,A -85,B 0,C 180,E1 -8013.506,E2 -8013.506} C_VEL
LIN {X 0,Y 459.617,Z 472.75,A -85,B 0,C 180,E1 -8014.823,E2 -8014.823} C_VEL
LIN {X 0,Y 459.673,Z 467.623,A -85,B 0,C 180,E1 -8016.386,E2 -8016.386} C_VEL
LIN {X 0,Y 459.865,Z 461.014,A -85,B 0,C 180,E1 -8017.905,E2 -8017.905} C_VEL
LIN {X 0,Y 460.098,Z 453.632,A -85,B 0,C 180,E1 -8019.228,E2 -8019.228} C_VEL
LIN {X 0,Y 460.437,Z 444.454,A -85,B 0,C 180,E1 -8020.553,E2 -8020.553} C_VEL
LIN {X 0,Y 460.939,Z 434.979,A -85,B 0,C 180,E1 -8021.654,E2 -8021.654} C_VEL
LIN {X 0,Y 461.322,Z 423.734,A -85,B 0,C 180,E1 -8022.753,E2 -8022.753} C_VEL
LIN {X 0,Y 461.918,Z 412.154,A -85,B 0,C 180,E1 -8023.639,E2 -8023.639} C_VEL
LIN {X 0,Y 462.424,Z 400.064,A -85,B 0,C 180,E1 -8024.353,E2 -8024.353} C_VEL
LIN {X 0,Y 462.921,Z 386.563,A -85,B 0,C 180,E1 -8024.928,E2 -8024.928} C_VEL
LIN {X 0,Y 463.296,Z 373.789,A -85,B 0,C 180,E1 -8025.281,E2 -8025.281} C_VEL
LIN {X 0,Y 463.944,Z 301.226,A -85,B 0,C 180,E1 -8026.472,E2 -8026.472} C_VEL
LIN {X 0,Y 463.936,Z 285.569,A -85,B 0,C 180,E1 -8026.758,E2 -8026.758} C_VEL
LIN {X 0,Y 461.299,Z 266.946,A -85,B 0,C 180,E1 -8027.208,E2 -8027.208} C_VEL
LIN {X 0,Y 462.036,Z 249.167,A -85,B 0,C 180,E1 -8030.245,E2 -8030.245} C_VEL
LIN {X 0,Y 462.891,Z 231.826,A -85,B 0,C 180,E1 -8033.249,E2 -8033.249} C_VEL
LIN {X 0,Y 463.123,Z 225.155,A -85,B 0,C 180,E1 -8034.423,E2 -8034.423} C_VEL
LIN {X 0,Y 460.613,Z 212.11,A -85,B 0,C 180,E1 -8036.903,E2 -8036.903} C_VEL
LIN {X 0,Y 460.507,Z 212.124,A -85,B 0,C 180,E1 -8040.239,E2 -8040.239} C_VEL
LIN {X 0,Y 460.525,Z 212.104,A -85,B 0,C 180,E1 -8043.324,E2 -8043.324} C_VEL
LIN {X 0,Y 460.468,Z 212.125,A -85,B 0,C 180,E1 -8046.529,E2 -8046.529} C_VEL
LIN {X 0,Y 460.508,Z 212.122,A -85,B 0,C 180,E1 -8049.863,E2 -8049.863} C_VEL
LIN {X 0,Y 460.486,Z 212.119,A -85,B 0,C 180,E1 -8052.897,E2 -8052.897} C_VEL
LIN {X 0,Y 460.497,Z 212.124,A -85,B 0,C 180,E1 -8055.831,E2 -8055.831} C_VEL
LIN {X 0,Y 460.511,Z 212.112,A -85,B 0,C 180,E1 -8058.987,E2 -8058.987} C_VEL
LIN {X 0,Y 460.493,Z 212.118,A -85,B 0,C 180,E1 -8062.376,E2 -8062.376} C_VEL
LIN {X 0,Y 460.529,Z 212.116,A -85,B 0,C 180,E1 -8065.622,E2 -8065.622} C_VEL
LIN {X 0,Y 460.529,Z 212.116,A -85,B 0,C 180,E1 -8068.744,E2 -8068.744} C_VEL
LIN {X 0,Y 460.498,Z 212.113,A -85,B 0,C 180,E1 -8071.763,E2 -8071.763} C_VEL
LIN {X 0,Y 460.511,Z 212.119,A -85,B 0,C 180,E1 -8074.703,E2 -8074.703} C_VEL
LIN {X 0,Y 460.497,Z 212.104,A -85,B 0,C 180,E1 -8077.571,E2 -8077.571} C_VEL
LIN {X 0,Y 460.554,Z 212.109,A -85,B 0,C 180,E1 -8080.384,E2 -8080.384} C_VEL
LIN {X 0,Y 460.569,Z 212.107,A -85,B 0,C 180,E1 -8084.012,E2 -8084.012} C_VEL
LIN {X 0,Y 460.599,Z 212.1,A -85,B 0,C 180,E1 -8087.666,E2 -8087.666} C_VEL
LIN {X 0,Y 460.606,Z 212.106,A -85,B 0,C 180,E1 -8091.224,E2 -8091.224} C_VEL
LIN {X 0,Y 460.65,Z 212.093,A -85,B 0,C 180,E1 -8093.869,E2 -8093.869} C_VEL
LIN {X 0,Y 460.778,Z 212.081,A -85,B 0,C 180,E1 -8097.378,E2 -8097.378} C_VEL
LIN {X 0,Y 460.809,Z 212.083,A -85,B 0,C 180,E1 -8100,E2 -8100} C_VEL
LIN {X 0,Y 460.756,Z 212.075,A -85,B 0,C 180,E1 -8102.623,E2 -8102.623} C_VEL
LIN {X 0,Y 460.692,Z 212.099,A -85,B 0,C 180,E1 -8106.13,E2 -8106.13} C_VEL
LIN {X 0,Y 460.618,Z 212.097,A -85,B 0,C 180,E1 -8108.777,E2 -8108.777} C_VEL
LIN {X 0,Y 460.605,Z 212.105,A -85,B 0,C 180,E1 -8112.445,E2 -8112.445} C_VEL
LIN {X 0,Y 460.592,Z 212.104,A -85,B 0,C 180,E1 -8115.998,E2 -8115.998} C_VEL
LIN {X 0,Y 460.561,Z 212.114,A -85,B 0,C 180,E1 -8119.616,E2 -8119.616} C_VEL
LIN {X 0,Y 460.504,Z 212.115,A -85,B 0,C 180,E1 -8122.429,E2 -8122.429} C_VEL
LIN {X 0,Y 460.561,Z 212.117,A -85,B 0,C 180,E1 -8125.803,E2 -8125.803} C_VEL
LIN {X 0,Y 460.545,Z 212.111,A -85,B 0,C 180,E1 -8128.234,E2 -8128.234} C_VEL
LIN {X 0,Y 460.515,Z 212.123,A -85,B 0,C 180,E1 -8131.284,E2 -8131.284} C_VEL
LIN {X 0,Y 460.528,Z 212.112,A -85,B 0,C 180,E1 -8134.507,E2 -8134.507} C_VEL
LIN {X 0,Y 460.524,Z 212.116,A -85,B 0,C 180,E1 -8137.622,E2 -8137.622} C_VEL
LIN {X 0,Y 460.538,Z 212.118,A -85,B 0,C 180,E1 -8140.271,E2 -8140.271} C_VEL
LIN {X 0,Y 460.504,Z 212.124,A -85,B 0,C 180,E1 -8143.375,E2 -8143.375} C_VEL
LIN {X 0,Y 460.505,Z 212.124,A -85,B 0,C 180,E1 -8146.627,E2 -8146.627} C_VEL
LIN {X 0,Y 460.539,Z 212.114,A -85,B 0,C 180,E1 -8149.732,E2 -8149.732} C_VEL
LIN {X 0,Y 460.498,Z 212.125,A -85,B 0,C 180,E1 -8152.525,E2 -8152.525} C_VEL
LIN {X 0,Y 460.546,Z 212.117,A -85,B 0,C 180,E1 -8155.625,E2 -8155.625} C_VEL
LIN {X 0,Y 460.645,Z 212.171,A -85,B 0,C 180,E1 -8157.445,E2 -8157.445} C_VEL
LIN {X 0,Y 461.243,Z 216.853,A -85,B 0,C 180,E1 -8157.997,E2 -8157.997} C_VEL
LIN {X 0,Y 461.419,Z 222.275,A -85,B 0,C 180,E1 -8158.606,E2 -8158.606} C_VEL
LIN {X 0,Y 464.856,Z 241.656,A -85,B 0,C 180,E1 -8159.068,E2 -8159.068} C_VEL
LIN {X 0,Y 463.967,Z 332.774,A -85,B 0,C 180,E1 -8160.51,E2 -8160.51} C_VEL
LIN {X 0,Y 463.667,Z 346.367,A -85,B 0,C 180,E1 -8160.893,E2 -8160.893} C_VEL
LIN {X 0,Y 463.364,Z 357.809,A -85,B 0,C 180,E1 -8161.381,E2 -8161.381} C_VEL
LIN {X 0,Y 463.021,Z 367.974,A -85,B 0,C 180,E1 -8161.953,E2 -8161.953} C_VEL
LIN {X 0,Y 462.13,Z 373.288,A -85,B 0,C 180,E1 -8162.284,E2 -8162.284} C_VEL
LIN {X 0,Y 457.487,Z 384.83,A -85,B 0,C 180,E1 -8163.059,E2 -8163.059} C_VEL
LIN {X 0,Y 455.262,Z 391.056,A -85,B 0,C 180,E1 -8163.594,E2 -8163.594} C_VEL
LIN {X 0,Y 454.802,Z 393.998,A -85,B 0,C 180,E1 -8163.902,E2 -8163.902} C_VEL
LIN {X 0,Y 454.287,Z 403.486,A -85,B 0,C 180,E1 -8165.068,E2 -8165.068} C_VEL
LIN {X 0,Y 453.808,Z 411.337,A -85,B 0,C 180,E1 -8166.257,E2 -8166.257} C_VEL
LIN {X 0,Y 453.334,Z 418.932,A -85,B 0,C 180,E1 -8167.679,E2 -8167.679} C_VEL
LIN {X 0,Y 453.033,Z 424.946,A -85,B 0,C 180,E1 -8169.097,E2 -8169.097} C_VEL
LIN {X 0,Y 452.773,Z 429.567,A -85,B 0,C 180,E1 -8170.506,E2 -8170.506} C_VEL
LIN {X 0,Y 452.633,Z 432.988,A -85,B 0,C 180,E1 -8171.909,E2 -8171.909} C_VEL
LIN {X 0,Y 452.527,Z 434.657,A -85,B 0,C 180,E1 -8172.839,E2 -8172.839} C_VEL
LIN {X 0,Y 452.444,Z 436.47,A -85,B 0,C 180,E1 -8174.383,E2 -8174.383} C_VEL
LIN {X 0,Y 452.419,Z 437.045,A -85,B 0,C 180,E1 -8175.609,E2 -8175.609} C_VEL
LIN {X 0,Y 452.394,Z 437.004,A -85,B 0,C 180,E1 -8176.526,E2 -8176.526} C_VEL
LIN {X 0,Y 452.516,Z 435.963,A -85,B 0,C 180,E1 -8178.086,E2 -8178.086} C_VEL
LIN {X 0,Y 452.539,Z 434.342,A -85,B 0,C 180,E1 -8179.261,E2 -8179.261} C_VEL
LIN {X 0,Y 452.643,Z 431.58,A -85,B 0,C 180,E1 -8180.618,E2 -8180.618} C_VEL
LIN {X 0,Y 452.807,Z 427.791,A -85,B 0,C 180,E1 -8181.971,E2 -8181.971} C_VEL
LIN {X 0,Y 453.051,Z 422.512,A -85,B 0,C 180,E1 -8183.411,E2 -8183.411} C_VEL
LIN {X 0,Y 453.383,Z 415.504,A -85,B 0,C 180,E1 -8184.887,E2 -8184.887} C_VEL
LIN {X 0,Y 453.747,Z 407.538,A -85,B 0,C 180,E1 -8186.227,E2 -8186.227} C_VEL
LIN {X 0,Y 454.206,Z 399.378,A -85,B 0,C 180,E1 -8187.34,E2 -8187.34} C_VEL
LIN {X 0,Y 454.709,Z 389.362,A -85,B 0,C 180,E1 -8188.451,E2 -8188.451} C_VEL
LIN {X 0,Y 455.336,Z 378.141,A -85,B 0,C 180,E1 -8189.448,E2 -8189.448} C_VEL
LIN {X 0,Y 455.832,Z 367.096,A -85,B 0,C 180,E1 -8190.222,E2 -8190.222} C_VEL
LIN {X 0,Y 456.207,Z 354.751,A -85,B 0,C 180,E1 -8190.884,E2 -8190.884} C_VEL
LIN {X 0,Y 456.589,Z 341.861,A -85,B 0,C 180,E1 -8191.379,E2 -8191.379} C_VEL
LIN {X 0,Y 456.767,Z 329.377,A -85,B 0,C 180,E1 -8191.682,E2 -8191.682} C_VEL
LIN {X 0,Y 457.481,Z 241.316,A -85,B 0,C 180,E1 -8193.07,E2 -8193.07} C_VEL
LIN {X 0,Y 454.127,Z 222.301,A -85,B 0,C 180,E1 -8193.5,E2 -8193.5} C_VEL
LIN {X 0,Y 453.735,Z 214.161,A -85,B 0,C 180,E1 -8194.443,E2 -8194.443} C_VEL
LIN {X 0,Y 453.527,Z 212.994,A -85,B 0,C 180,E1 -8194.612,E2 -8194.612} C_VEL
LIN {X 0,Y 453.664,Z 212.974,A -85,B 0,C 180,E1 -8196.226,E2 -8196.226} C_VEL
LIN {X 0,Y 453.589,Z 212.985,A -85,B 0,C 180,E1 -8198.914,E2 -8198.914} C_VEL
LIN {X 0,Y 453.571,Z 212.986,A -85,B 0,C 180,E1 -8202.53,E2 -8202.53} C_VEL
LIN {X 0,Y 453.551,Z 212.988,A -85,B 0,C 180,E1 -8206.197,E2 -8206.197} C_VEL
LIN {X 0,Y 453.523,Z 212.993,A -85,B 0,C 180,E1 -8209.04,E2 -8209.04} C_VEL
LIN {X 0,Y 453.482,Z 212.997,A -85,B 0,C 180,E1 -8211.837,E2 -8211.837} C_VEL
LIN {X 0,Y 453.474,Z 212.999,A -85,B 0,C 180,E1 -8214.738,E2 -8214.738} C_VEL
LIN {X 0,Y 453.469,Z 212.998,A -85,B 0,C 180,E1 -8217.943,E2 -8217.943} C_VEL
LIN {X 0,Y 453.463,Z 213,A -85,B 0,C 180,E1 -8220.761,E2 -8220.761} C_VEL
LIN {X 0,Y 453.472,Z 212.998,A -85,B 0,C 180,E1 -8223.914,E2 -8223.914} C_VEL
LIN {X 0,Y 453.444,Z 213.002,A -85,B 0,C 180,E1 -8227.192,E2 -8227.192} C_VEL
LIN {X 0,Y 453.472,Z 212.999,A -85,B 0,C 180,E1 -8230.612,E2 -8230.612} C_VEL
LIN {X 0,Y 453.482,Z 212.997,A -85,B 0,C 180,E1 -8234.528,E2 -8234.528} C_VEL
LIN {X 0,Y 453.436,Z 213.004,A -85,B 0,C 180,E1 -8238.072,E2 -8238.072} C_VEL
LIN {X 0,Y 453.427,Z 213.005,A -85,B 0,C 180,E1 -8240.805,E2 -8240.805} C_VEL
LIN {X 0,Y 453.419,Z 213.006,A -85,B 0,C 180,E1 -8243.913,E2 -8243.913} C_VEL
LIN {X 0,Y 453.46,Z 213,A -85,B 0,C 180,E1 -8247.149,E2 -8247.149} C_VEL
LIN {X 0,Y 453.453,Z 213.002,A -85,B 0,C 180,E1 -8250.266,E2 -8250.266} C_VEL
LIN {X 0,Y 453.429,Z 213.005,A -85,B 0,C 180,E1 -8253.289,E2 -8253.289} C_VEL
LIN {X 0,Y 453.498,Z 212.997,A -85,B 0,C 180,E1 -8256.238,E2 -8256.238} C_VEL
LIN {X 0,Y 453.528,Z 213.079,A -85,B 0,C 180,E1 -8258.519,E2 -8258.519} C_VEL
LIN {X 0,Y 454.615,Z 219.805,A -85,B 0,C 180,E1 -8260.116,E2 -8260.116} C_VEL
LIN {X 0,Y 454.467,Z 226.704,A -85,B 0,C 180,E1 -8261.677,E2 -8261.677} C_VEL
LIN {X 0,Y 457.453,Z 242.471,A -85,B 0,C 180,E1 -8262.084,E2 -8262.084} C_VEL
LIN {X 0,Y 456.21,Z 334.06,A -85,B 0,C 180,E1 -8263.757,E2 -8263.757} C_VEL
LIN {X 0,Y 455.956,Z 346.725,A -85,B 0,C 180,E1 -8264.15,E2 -8264.15} C_VEL
LIN {X 0,Y 455.612,Z 359.832,A -85,B 0,C 180,E1 -8264.74,E2 -8264.74} C_VEL
LIN {X 0,Y 455.158,Z 371.765,A -85,B 0,C 180,E1 -8265.468,E2 -8265.468} C_VEL
LIN {X 0,Y 454.677,Z 383.278,A -85,B 0,C 180,E1 -8266.366,E2 -8266.366} C_VEL
LIN {X 0,Y 454.283,Z 393.485,A -85,B 0,C 180,E1 -8267.357,E2 -8267.357} C_VEL
LIN {X 0,Y 453.914,Z 402.164,A -85,B 0,C 180,E1 -8268.388,E2 -8268.388} C_VEL
LIN {X 0,Y 453.452,Z 411.38,A -85,B 0,C 180,E1 -8269.733,E2 -8269.733} C_VEL
LIN {X 0,Y 453.16,Z 418.794,A -85,B 0,C 180,E1 -8271.078,E2 -8271.078} C_VEL
LIN {X 0,Y 452.893,Z 424.685,A -85,B 0,C 180,E1 -8272.42,E2 -8272.42} C_VEL
LIN {X 0,Y 452.79,Z 429.303,A -85,B 0,C 180,E1 -8273.762,E2 -8273.762} C_VEL
LIN {X 0,Y 452.687,Z 431.739,A -85,B 0,C 180,E1 -8274.655,E2 -8274.655} C_VEL
LIN {X 0,Y 452.587,Z 433.735,A -85,B 0,C 180,E1 -8275.547,E2 -8275.547} C_VEL
LIN {X 0,Y 452.66,Z 435.262,A -85,B 0,C 180,E1 -8276.439,E2 -8276.439} C_VEL
LIN {X 0,Y 452.582,Z 436.348,A -85,B 0,C 180,E1 -8277.33,E2 -8277.33} C_VEL
LIN {X 0,Y 452.52,Z 437.032,A -85,B 0,C 180,E1 -8278.22,E2 -8278.22} C_VEL
LIN {X 0,Y 452.499,Z 437.31,A -85,B 0,C 180,E1 -8279.11,E2 -8279.11} C_VEL
LIN {X 0,Y 452.478,Z 437.134,A -85,B 0,C 180,E1 -8280,E2 -8280} C_VEL
LIN {X 0,Y 452.504,Z 436.547,A -85,B 0,C 180,E1 -8280.89,E2 -8280.89} C_VEL
LIN {X 0,Y 452.592,Z 435.556,A -85,B 0,C 180,E1 -8281.78,E2 -8281.78} C_VEL
LIN {X 0,Y 452.746,Z 434.131,A -85,B 0,C 180,E1 -8282.669,E2 -8282.669} C_VEL
LIN {X 0,Y 452.821,Z 431.152,A -85,B 0,C 180,E1 -8284.005,E2 -8284.005} C_VEL
LIN {X 0,Y 452.915,Z 427.091,A -85,B 0,C 180,E1 -8285.342,E2 -8285.342} C_VEL
LIN {X 0,Y 453.276,Z 421.241,A -85,B 0,C 180,E1 -8286.805,E2 -8286.805} C_VEL
LIN {X 0,Y 453.559,Z 413.961,A -85,B 0,C 180,E1 -8288.24,E2 -8288.24} C_VEL
LIN {X 0,Y 453.96,Z 406.943,A -85,B 0,C 180,E1 -8289.355,E2 -8289.355} C_VEL
LIN {X 0,Y 454.355,Z 398.473,A -85,B 0,C 180,E1 -8290.472,E2 -8290.472} C_VEL
LIN {X 0,Y 454.824,Z 387.996,A -85,B 0,C 180,E1 -8291.588,E2 -8291.588} C_VEL
LIN {X 0,Y 455.4,Z 377.655,A -85,B 0,C 180,E1 -8292.477,E2 -8292.477} C_VEL
LIN {X 0,Y 455.821,Z 366.367,A -85,B 0,C 180,E1 -8293.259,E2 -8293.259} C_VEL
LIN {X 0,Y 456.307,Z 353.241,A -85,B 0,C 180,E1 -8293.94,E2 -8293.94} C_VEL
LIN {X 0,Y 456.568,Z 340.209,A -85,B 0,C 180,E1 -8294.429,E2 -8294.429} C_VEL
LIN {X 0,Y 456.858,Z 324.102,A -85,B 0,C 180,E1 -8294.789,E2 -8294.789} C_VEL
LIN {X 0,Y 458.361,Z 245.703,A -85,B 0,C 180,E1 -8296.324,E2 -8296.324} C_VEL
LIN {X 0,Y 458.187,Z 241.909,A -85,B 0,C 180,E1 -8296.414,E2 -8296.414} C_VEL
LIN {X 0,Y 455.314,Z 229.496,A -85,B 0,C 180,E1 -8296.836,E2 -8296.836} C_VEL
LIN {X 0,Y 455.434,Z 223.075,A -85,B 0,C 180,E1 -8298.442,E2 -8298.442} C_VEL
LIN {X 0,Y 454.203,Z 215.991,A -85,B 0,C 180,E1 -8300.374,E2 -8300.374} C_VEL
LIN {X 0,Y 453.501,Z 212.999,A -85,B 0,C 180,E1 -8301.274,E2 -8301.274} C_VEL
LIN {X 0,Y 453.506,Z 212.998,A -85,B 0,C 180,E1 -8304.735,E2 -8304.735} C_VEL
LIN {X 0,Y 453.538,Z 212.992,A -85,B 0,C 180,E1 -8307.959,E2 -8307.959} C_VEL
LIN {X 0,Y 453.471,Z 212.998,A -85,B 0,C 180,E1 -8311.525,E2 -8311.525} C_VEL
LIN {X 0,Y 453.493,Z 212.996,A -85,B 0,C 180,E1 -8314.777,E2 -8314.777} C_VEL
LIN {X 0,Y 453.469,Z 213.002,A -85,B 0,C 180,E1 -8318.311,E2 -8318.311} C_VEL
LIN {X 0,Y 453.499,Z 212.995,A -85,B 0,C 180,E1 -8320.608,E2 -8320.608} C_VEL
LIN {X 0,Y 453.458,Z 212.999,A -85,B 0,C 180,E1 -8323.243,E2 -8323.243} C_VEL
LIN {X 0,Y 453.465,Z 213,A -85,B 0,C 180,E1 -8325.778,E2 -8325.778} C_VEL
LIN {X 0,Y 453.498,Z 212.995,A -85,B 0,C 180,E1 -8329.409,E2 -8329.409} C_VEL
LIN {X 0,Y 453.454,Z 213,A -85,B 0,C 180,E1 -8332.809,E2 -8332.809} C_VEL
LIN {X 0,Y 453.481,Z 213.002,A -85,B 0,C 180,E1 -8336.087,E2 -8336.087} C_VEL
LIN {X 0,Y 453.48,Z 213.004,A -85,B 0,C 180,E1 -8339.24,E2 -8339.24} C_VEL
LIN {X 0,Y 453.527,Z 213.062,A -85,B 0,C 180,E1 -8342.176,E2 -8342.176} C_VEL
LIN {X 0,Y 455.776,Z 223.097,A -85,B 0,C 180,E1 -8344.42,E2 -8344.42} C_VEL
LIN {X 0,Y 456.605,Z 228.002,A -85,B 0,C 180,E1 -8345.443,E2 -8345.443} C_VEL
LIN {X 0,Y 455.648,Z 243.103,A -85,B 0,C 180,E1 -8348.272,E2 -8348.272} C_VEL
LIN {X 0,Y 454.579,Z 262.407,A -85,B 0,C 180,E1 -8351.754,E2 -8351.754} C_VEL
LIN {X 0,Y 454.472,Z 264.506,A -85,B 0,C 180,E1 -8352.127,E2 -8352.127} C_VEL
LIN {X 0,Y 457.323,Z 282.943,A -85,B 0,C 180,E1 -8352.666,E2 -8352.666} C_VEL
LIN {X 0,Y 457.822,Z 288.91,A -85,B 0,C 180,E1 -8352.815,E2 -8352.815} C_VEL
LIN {X 0,Y 456.654,Z 360.639,A -85,B 0,C 180,E1 -8354.203,E2 -8354.203} C_VEL
LIN {X 0,Y 456.331,Z 377.654,A -85,B 0,C 180,E1 -8354.564,E2 -8354.564} C_VEL
LIN {X 0,Y 455.891,Z 391.116,A -85,B 0,C 180,E1 -8355.035,E2 -8355.035} C_VEL
LIN {X 0,Y 455.317,Z 404.464,A -85,B 0,C 180,E1 -8355.701,E2 -8355.701} C_VEL
LIN {X 0,Y 454.783,Z 416.305,A -85,B 0,C 180,E1 -8356.482,E2 -8356.482} C_VEL
LIN {X 0,Y 454.202,Z 428.233,A -85,B 0,C 180,E1 -8357.488,E2 -8357.488} C_VEL
LIN {X 0,Y 453.716,Z 438.865,A -85,B 0,C 180,E1 -8358.608,E2 -8358.608} C_VEL
LIN {X 0,Y 453.188,Z 449.038,A -85,B 0,C 180,E1 -8359.952,E2 -8359.952} C_VEL
LIN {X 0,Y 452.913,Z 457.235,A -85,B 0,C 180,E1 -8361.297,E2 -8361.297} C_VEL
LIN {X 0,Y 452.728,Z 462.793,A -85,B 0,C 180,E1 -8362.417,E2 -8362.417} C_VEL
LIN {X 0,Y 452.564,Z 468.21,A -85,B 0,C 180,E1 -8363.758,E2 -8363.758} C_VEL
LIN {X 0,Y 452.544,Z 472.417,A -85,B 0,C 180,E1 -8365.099,E2 -8365.099} C_VEL
LIN {X 0,Y 452.492,Z 475.529,A -85,B 0,C 180,E1 -8366.437,E2 -8366.437} C_VEL
LIN {X 0,Y 452.524,Z 477.012,A -85,B 0,C 180,E1 -8367.329,E2 -8367.329} C_VEL
LIN {X 0,Y 452.483,Z 478.072,A -85,B 0,C 180,E1 -8368.219,E2 -8368.219} C_VEL
LIN {X 0,Y 452.491,Z 478.724,A -85,B 0,C 180,E1 -8369.109,E2 -8369.109} C_VEL
LIN {X 0,Y 452.471,Z 478.931,A -85,B 0,C 180,E1 -8369.999,E2 -8369.999} C_VEL
LIN {X 0,Y 452.491,Z 478.696,A -85,B 0,C 180,E1 -8370.889,E2 -8370.889} C_VEL
LIN {X 0,Y 452.483,Z 478.05,A -85,B 0,C 180,E1 -8371.779,E2 -8371.779} C_VEL
LIN {X 0,Y 452.527,Z 476.994,A -85,B 0,C 180,E1 -8372.669,E2 -8372.669} C_VEL
LIN {X 0,Y 452.521,Z 475.459,A -85,B 0,C 180,E1 -8373.561,E2 -8373.561} C_VEL
LIN {X 0,Y 452.547,Z 472.323,A -85,B 0,C 180,E1 -8374.899,E2 -8374.899} C_VEL
LIN {X 0,Y 452.569,Z 467.662,A -85,B 0,C 180,E1 -8376.35,E2 -8376.35} C_VEL
LIN {X 0,Y 452.755,Z 461.551,A -85,B 0,C 180,E1 -8377.805,E2 -8377.805} C_VEL
LIN {X 0,Y 453.003,Z 454.419,A -85,B 0,C 180,E1 -8379.149,E2 -8379.149} C_VEL
LIN {X 0,Y 453.319,Z 445.495,A -85,B 0,C 180,E1 -8380.495,E2 -8380.495} C_VEL
LIN {X 0,Y 453.821,Z 436.794,A -85,B 0,C 180,E1 -8381.613,E2 -8381.613} C_VEL
LIN {X 0,Y 454.253,Z 427.094,A -85,B 0,C 180,E1 -8382.636,E2 -8382.636} C_VEL
LIN {X 0,Y 454.804,Z 416.81,A -85,B 0,C 180,E1 -8383.515,E2 -8383.515} C_VEL
LIN {X 0,Y 455.37,Z 405.271,A -85,B 0,C 180,E1 -8384.295,E2 -8384.295} C_VEL
LIN {X 0,Y 455.847,Z 393.263,A -85,B 0,C 180,E1 -8384.908,E2 -8384.908} C_VEL
LIN {X 0,Y 456.364,Z 380.185,A -85,B 0,C 180,E1 -8385.376,E2 -8385.376} C_VEL
LIN {X 0,Y 456.594,Z 367.43,A -85,B 0,C 180,E1 -8385.654,E2 -8385.654} C_VEL
LIN {X 0,Y 457.12,Z 286.745,A -85,B 0,C 180,E1 -8386.957,E2 -8386.957} C_VEL
LIN {X 0,Y 454.325,Z 266.679,A -85,B 0,C 180,E1 -8387.452,E2 -8387.452} C_VEL
LIN {X 0,Y 455.046,Z 250.084,A -85,B 0,C 180,E1 -8390.334,E2 -8390.334} C_VEL
LIN {X 0,Y 455.946,Z 232.72,A -85,B 0,C 180,E1 -8393.384,E2 -8393.384} C_VEL
LIN {X 0,Y 456.079,Z 225.879,A -85,B 0,C 180,E1 -8394.609,E2 -8394.609} C_VEL
LIN {X 0,Y 453.571,Z 212.987,A -85,B 0,C 180,E1 -8397.136,E2 -8397.136} C_VEL
LIN {X 0,Y 453.473,Z 212.996,A -85,B 0,C 180,E1 -8400.758,E2 -8400.758} C_VEL
LIN {X 0,Y 453.472,Z 212.981,A -85,B 0,C 180,E1 -8403.912,E2 -8403.912} C_VEL
LIN {X 0,Y 453.444,Z 213,A -85,B 0,C 180,E1 -8407.189,E2 -8407.189} C_VEL
LIN {X 0,Y 453.465,Z 212.996,A -85,B 0,C 180,E1 -8410.611,E2 -8410.611} C_VEL
LIN {X 0,Y 453.454,Z 212.997,A -85,B 0,C 180,E1 -8414.221,E2 -8414.221} C_VEL
LIN {X 0,Y 453.43,Z 213.002,A -85,B 0,C 180,E1 -8417.001,E2 -8417.001} C_VEL
LIN {X 0,Y 453.463,Z 212.995,A -85,B 0,C 180,E1 -8419.412,E2 -8419.412} C_VEL
LIN {X 0,Y 453.444,Z 212.998,A -85,B 0,C 180,E1 -8422.81,E2 -8422.81} C_VEL
LIN {X 0,Y 453.46,Z 212.994,A -85,B 0,C 180,E1 -8426.086,E2 -8426.086} C_VEL
LIN {X 0,Y 453.465,Z 212.991,A -85,B 0,C 180,E1 -8429.24,E2 -8429.24} C_VEL
LIN {X 0,Y 453.465,Z 212.988,A -85,B 0,C 180,E1 -8432.293,E2 -8432.293} C_VEL
LIN {X 0,Y 453.458,Z 212.995,A -85,B 0,C 180,E1 -8435.262,E2 -8435.262} C_VEL
LIN {X 0,Y 453.471,Z 212.98,A -85,B 0,C 180,E1 -8438.415,E2 -8438.415} C_VEL
LIN {X 0,Y 453.513,Z 212.994,A -85,B 0,C 180,E1 -8441.008,E2 -8441.008} C_VEL
LIN {X 0,Y 453.528,Z 212.984,A -85,B 0,C 180,E1 -8443.893,E2 -8443.893} C_VEL
LIN {X 0,Y 453.555,Z 212.978,A -85,B 0,C 180,E1 -8447.471,E2 -8447.471} C_VEL
LIN {X 0,Y 453.572,Z 212.983,A -85,B 0,C 180,E1 -8451.086,E2 -8451.086} C_VEL
LIN {X 0,Y 453.619,Z 212.968,A -85,B 0,C 180,E1 -8453.774,E2 -8453.774} C_VEL
LIN {X 0,Y 453.722,Z 212.96,A -85,B 0,C 180,E1 -8457.337,E2 -8457.337} C_VEL
LIN {X 0,Y 453.779,Z 212.959,A -85,B 0,C 180,E1 -8460,E2 -8460} C_VEL
LIN {X 0,Y 453.703,Z 212.952,A -85,B 0,C 180,E1 -8462.664,E2 -8462.664} C_VEL
LIN {X 0,Y 453.66,Z 212.975,A -85,B 0,C 180,E1 -8466.226,E2 -8466.226} C_VEL
LIN {X 0,Y 453.581,Z 212.973,A -85,B 0,C 180,E1 -8468.914,E2 -8468.914} C_VEL
LIN {X 0,Y 453.555,Z 212.983,A -85,B 0,C 180,E1 -8472.529,E2 -8472.529} C_VEL
LIN {X 0,Y 453.536,Z 212.98,A -85,B 0,C 180,E1 -8476.197,E2 -8476.197} C_VEL
LIN {X 0,Y 453.509,Z 212.986,A -85,B 0,C 180,E1 -8479.04,E2 -8479.04} C_VEL
LIN {X 0,Y 453.469,Z 212.996,A -85,B 0,C 180,E1 -8481.837,E2 -8481.837} C_VEL
LIN {X 0,Y 453.507,Z 212.985,A -85,B 0,C 180,E1 -8484.735,E2 -8484.735} C_VEL
LIN {X 0,Y 453.525,Z 212.987,A -85,B 0,C 180,E1 -8487.96,E2 -8487.96} C_VEL
LIN {X 0,Y 453.46,Z 213.003,A -85,B 0,C 180,E1 -8491.526,E2 -8491.526} C_VEL
LIN {X 0,Y 453.483,Z 212.991,A -85,B 0,C 180,E1 -8494.779,E2 -8494.779} C_VEL
LIN {X 0,Y 453.469,Z 212.993,A -85,B 0,C 180,E1 -8498.312,E2 -8498.312} C_VEL
LIN {X 0,Y 453.49,Z 212.998,A -85,B 0,C 180,E1 -8500.61,E2 -8500.61} C_VEL
LIN {X 0,Y 453.469,Z 212.997,A -85,B 0,C 180,E1 -8504.221,E2 -8504.221} C_VEL
LIN {X 0,Y 453.465,Z 213,A -85,B 0,C 180,E1 -8507.007,E2 -8507.007} C_VEL
LIN {X 0,Y 453.503,Z 212.995,A -85,B 0,C 180,E1 -8510.553,E2 -8510.553} C_VEL
LIN {X 0,Y 453.453,Z 213,A -85,B 0,C 180,E1 -8513.918,E2 -8513.918} C_VEL
LIN {X 0,Y 453.605,Z 213.153,A -85,B 0,C 180,E1 -8517.245,E2 -8517.245} C_VEL
LIN {X 0,Y 454.384,Z 217.405,A -85,B 0,C 180,E1 -8517.752,E2 -8517.752} C_VEL
LIN {X 0,Y 454.556,Z 222.196,A -85,B 0,C 180,E1 -8518.287,E2 -8518.287} C_VEL
LIN {X 0,Y 458.113,Z 241.636,A -85,B 0,C 180,E1 -8518.777,E2 -8518.777} C_VEL
LIN {X 0,Y 457.199,Z 333.286,A -85,B 0,C 180,E1 -8520.251,E2 -8520.251} C_VEL
LIN {X 0,Y 456.889,Z 346.824,A -85,B 0,C 180,E1 -8520.64,E2 -8520.64} C_VEL
LIN {X 0,Y 456.528,Z 359.465,A -85,B 0,C 180,E1 -8521.202,E2 -8521.202} C_VEL
LIN {X 0,Y 456.016,Z 372.084,A -85,B 0,C 180,E1 -8521.963,E2 -8521.963} C_VEL
LIN {X 0,Y 455.428,Z 382.797,A -85,B 0,C 180,E1 -8522.797,E2 -8522.797} C_VEL
LIN {X 0,Y 454.802,Z 393.998,A -85,B 0,C 180,E1 -8523.902,E2 -8523.902} C_VEL
LIN {X 0,Y 453.931,Z 398.41,A -85,B 0,C 180,E1 -8524.386,E2 -8524.386} C_VEL
LIN {X 0,Y 450.743,Z 405.311,A -85,B 0,C 180,E1 -8525.194,E2 -8525.194} C_VEL
LIN {X 0,Y 447.53,Z 411.609,A -85,B 0,C 180,E1 -8526.081,E2 -8526.081} C_VEL
LIN {X 0,Y 446.63,Z 415.074,A -85,B 0,C 180,E1 -8526.684,E2 -8526.684} C_VEL
LIN {X 0,Y 446.198,Z 421.944,A -85,B 0,C 180,E1 -8528.124,E2 -8528.124} C_VEL
LIN {X 0,Y 445.839,Z 427.844,A -85,B 0,C 180,E1 -8529.71,E2 -8529.71} C_VEL
LIN {X 0,Y 445.658,Z 431.771,A -85,B 0,C 180,E1 -8531.121,E2 -8531.121} C_VEL
LIN {X 0,Y 445.463,Z 434.659,A -85,B 0,C 180,E1 -8532.558,E2 -8532.558} C_VEL
LIN {X 0,Y 445.37,Z 436.742,A -85,B 0,C 180,E1 -8534.28,E2 -8534.28} C_VEL
LIN {X 0,Y 445.337,Z 437.327,A -85,B 0,C 180,E1 -8535.376,E2 -8535.376} C_VEL
LIN {X 0,Y 445.307,Z 437.354,A -85,B 0,C 180,E1 -8536.307,E2 -8536.307} C_VEL
LIN {X 0,Y 445.43,Z 436.341,A -85,B 0,C 180,E1 -8538.027,E2 -8538.027} C_VEL
LIN {X 0,Y 445.436,Z 434.967,A -85,B 0,C 180,E1 -8539.087,E2 -8539.087} C_VEL
LIN {X 0,Y 445.532,Z 432.347,A -85,B 0,C 180,E1 -8540.467,E2 -8540.467} C_VEL
LIN {X 0,Y 445.707,Z 428.704,A -85,B 0,C 180,E1 -8541.842,E2 -8541.842} C_VEL
LIN {X 0,Y 445.983,Z 423.204,A -85,B 0,C 180,E1 -8543.404,E2 -8543.404} C_VEL
LIN {X 0,Y 446.274,Z 416.835,A -85,B 0,C 180,E1 -8544.806,E2 -8544.806} C_VEL
LIN {X 0,Y 446.673,Z 409.06,A -85,B 0,C 180,E1 -8546.167,E2 -8546.167} C_VEL
LIN {X 0,Y 447.127,Z 401.141,A -85,B 0,C 180,E1 -8547.298,E2 -8547.298} C_VEL
LIN {X 0,Y 447.645,Z 391.536,A -85,B 0,C 180,E1 -8548.427,E2 -8548.427} C_VEL
LIN {X 0,Y 448.265,Z 380.731,A -85,B 0,C 180,E1 -8549.44,E2 -8549.44} C_VEL
LIN {X 0,Y 448.858,Z 368.595,A -85,B 0,C 180,E1 -8550.337,E2 -8550.337} C_VEL
LIN {X 0,Y 449.236,Z 356.681,A -85,B 0,C 180,E1 -8551.009,E2 -8551.009} C_VEL
LIN {X 0,Y 449.636,Z 343.582,A -85,B 0,C 180,E1 -8551.54,E2 -8551.54} C_VEL
LIN {X 0,Y 449.854,Z 330.803,A -85,B 0,C 180,E1 -8551.876,E2 -8551.876} C_VEL
LIN {X 0,Y 450.631,Z 241.962,A -85,B 0,C 180,E1 -8553.298,E2 -8553.298} C_VEL
LIN {X 0,Y 447.155,Z 222.149,A -85,B 0,C 180,E1 -8553.775,E2 -8553.775} C_VEL
LIN {X 0,Y 446.659,Z 214.688,A -85,B 0,C 180,E1 -8554.626,E2 -8554.626} C_VEL
LIN {X 0,Y 446.501,Z 213.87,A -85,B 0,C 180,E1 -8554.741,E2 -8554.741} C_VEL
LIN {X 0,Y 446.634,Z 213.85,A -85,B 0,C 180,E1 -8556.325,E2 -8556.325} C_VEL
LIN {X 0,Y 446.537,Z 213.865,A -85,B 0,C 180,E1 -8559.056,E2 -8559.056} C_VEL
LIN {X 0,Y 446.528,Z 213.865,A -85,B 0,C 180,E1 -8562.73,E2 -8562.73} C_VEL
LIN {X 0,Y 446.495,Z 213.868,A -85,B 0,C 180,E1 -8566.46,E2 -8566.46} C_VEL
LIN {X 0,Y 446.475,Z 213.87,A -85,B 0,C 180,E1 -8569.304,E2 -8569.304} C_VEL
LIN {X 0,Y 446.423,Z 213.876,A -85,B 0,C 180,E1 -8572.2,E2 -8572.2} C_VEL
LIN {X 0,Y 446.426,Z 213.876,A -85,B 0,C 180,E1 -8575.155,E2 -8575.155} C_VEL
LIN {X 0,Y 446.443,Z 213.875,A -85,B 0,C 180,E1 -8578.182,E2 -8578.182} C_VEL
LIN {X 0,Y 446.414,Z 213.879,A -85,B 0,C 180,E1 -8581.301,E2 -8581.301} C_VEL
LIN {X 0,Y 446.427,Z 213.876,A -85,B 0,C 180,E1 -8584.524,E2 -8584.524} C_VEL
LIN {X 0,Y 446.402,Z 213.881,A -85,B 0,C 180,E1 -8588.076,E2 -8588.076} C_VEL
LIN {X 0,Y 446.401,Z 213.879,A -85,B 0,C 180,E1 -8591.395,E2 -8591.395} C_VEL
LIN {X 0,Y 446.423,Z 213.877,A -85,B 0,C 180,E1 -8595.109,E2 -8595.109} C_VEL
LIN {X 0,Y 446.4,Z 213.88,A -85,B 0,C 180,E1 -8598.605,E2 -8598.605} C_VEL
LIN {X 0,Y 446.39,Z 213.881,A -85,B 0,C 180,E1 -8602.119,E2 -8602.119} C_VEL
LIN {X 0,Y 446.388,Z 213.882,A -85,B 0,C 180,E1 -8605.473,E2 -8605.473} C_VEL
LIN {X 0,Y 446.395,Z 213.88,A -85,B 0,C 180,E1 -8608.698,E2 -8608.698} C_VEL
LIN {X 0,Y 446.407,Z 213.879,A -85,B 0,C 180,E1 -8611.842,E2 -8611.842} C_VEL
LIN {X 0,Y 446.419,Z 213.877,A -85,B 0,C 180,E1 -8614.845,E2 -8614.845} C_VEL
LIN {X 0,Y 446.499,Z 214.015,A -85,B 0,C 180,E1 -8618.393,E2 -8618.393} C_VEL
LIN {X 0,Y 447.625,Z 221.434,A -85,B 0,C 180,E1 -8620.171,E2 -8620.171} C_VEL
LIN {X 0,Y 447.489,Z 226.954,A -85,B 0,C 180,E1 -8621.433,E2 -8621.433} C_VEL
LIN {X 0,Y 450.578,Z 243.957,A -85,B 0,C 180,E1 -8621.88,E2 -8621.88} C_VEL
LIN {X 0,Y 449.249,Z 334.819,A -85,B 0,C 180,E1 -8623.586,E2 -8623.586} C_VEL
LIN {X 0,Y 448.988,Z 348.052,A -85,B 0,C 180,E1 -8624.014,E2 -8624.014} C_VEL
LIN {X 0,Y 448.646,Z 360.83,A -85,B 0,C 180,E1 -8624.613,E2 -8624.613} C_VEL
LIN {X 0,Y 448.155,Z 372.601,A -85,B 0,C 180,E1 -8625.352,E2 -8625.352} C_VEL
LIN {X 0,Y 447.673,Z 384.027,A -85,B 0,C 180,E1 -8626.264,E2 -8626.264} C_VEL
LIN {X 0,Y 447.236,Z 394.327,A -85,B 0,C 180,E1 -8627.291,E2 -8627.291} C_VEL
LIN {X 0,Y 446.813,Z 403.605,A -85,B 0,C 180,E1 -8628.431,E2 -8628.431} C_VEL
LIN {X 0,Y 446.397,Z 412.653,A -85,B 0,C 180,E1 -8629.798,E2 -8629.798} C_VEL
LIN {X 0,Y 446.06,Z 419.854,A -85,B 0,C 180,E1 -8631.163,E2 -8631.163} C_VEL
LIN {X 0,Y 445.778,Z 426.433,A -85,B 0,C 180,E1 -8632.754,E2 -8632.754} C_VEL
LIN {X 0,Y 445.693,Z 430.738,A -85,B 0,C 180,E1 -8634.117,E2 -8634.117} C_VEL
LIN {X 0,Y 445.506,Z 433.939,A -85,B 0,C 180,E1 -8635.476,E2 -8635.476} C_VEL
LIN {X 0,Y 445.573,Z 435.516,A -85,B 0,C 180,E1 -8636.382,E2 -8636.382} C_VEL
LIN {X 0,Y 445.509,Z 436.626,A -85,B 0,C 180,E1 -8637.287,E2 -8637.287} C_VEL
LIN {X 0,Y 445.435,Z 437.336,A -85,B 0,C 180,E1 -8638.191,E2 -8638.191} C_VEL
LIN {X 0,Y 445.419,Z 437.643,A -85,B 0,C 180,E1 -8639.096,E2 -8639.096} C_VEL
LIN {X 0,Y 445.413,Z 437.501,A -85,B 0,C 180,E1 -8640,E2 -8640} C_VEL
LIN {X 0,Y 445.442,Z 436.932,A -85,B 0,C 180,E1 -8640.904,E2 -8640.904} C_VEL
LIN {X 0,Y 445.535,Z 435.959,A -85,B 0,C 180,E1 -8641.808,E2 -8641.808} C_VEL
LIN {X 0,Y 445.677,Z 434.566,A -85,B 0,C 180,E1 -8642.711,E2 -8642.711} C_VEL
LIN {X 0,Y 445.767,Z 431.619,A -85,B 0,C 180,E1 -8644.068,E2 -8644.068} C_VEL
LIN {X 0,Y 445.856,Z 427.599,A -85,B 0,C 180,E1 -8645.427,E2 -8645.427} C_VEL
LIN {X 0,Y 446.235,Z 422.091,A -85,B 0,C 180,E1 -8646.845,E2 -8646.845} C_VEL
LIN {X 0,Y 446.577,Z 414.537,A -85,B 0,C 180,E1 -8648.37,E2 -8648.37} C_VEL
LIN {X 0,Y 447.119,Z 406.01,A -85,B 0,C 180,E1 -8649.728,E2 -8649.728} C_VEL
LIN {X 0,Y 447.568,Z 397.236,A -85,B 0,C 180,E1 -8650.861,E2 -8650.861} C_VEL
LIN {X 0,Y 448.092,Z 387.606,A -85,B 0,C 180,E1 -8651.879,E2 -8651.879} C_VEL
LIN {X 0,Y 448.635,Z 377.116,A -85,B 0,C 180,E1 -8652.784,E2 -8652.784} C_VEL
LIN {X 0,Y 449.072,Z 365.533,A -85,B 0,C 180,E1 -8653.577,E2 -8653.577} C_VEL
LIN {X 0,Y 449.567,Z 352.602,A -85,B 0,C 180,E1 -8654.246,E2 -8654.246} C_VEL
LIN {X 0,Y 449.837,Z 340.28,A -85,B 0,C 180,E1 -8654.707,E2 -8654.707} C_VEL
LIN {X 0,Y 450.143,Z 324.193,A -85,B 0,C 180,E1 -8655.073,E2 -8655.073} C_VEL
LIN {X 0,Y 451.805,Z 244.843,A -85,B 0,C 180,E1 -8656.68,E2 -8656.68} C_VEL
LIN {X 0,Y 449.609,Z 234.276,A -85,B 0,C 180,E1 -8657.038,E2 -8657.038} C_VEL
LIN {X 0,Y 448.505,Z 229.975,A -85,B 0,C 180,E1 -8657.204,E2 -8657.204} C_VEL
LIN {X 0,Y 448.472,Z 224.03,A -85,B 0,C 180,E1 -8658.739,E2 -8658.739} C_VEL
LIN {X 0,Y 447.196,Z 217.04,A -85,B 0,C 180,E1 -8660.708,E2 -8660.708} C_VEL
LIN {X 0,Y 446.453,Z 213.876,A -85,B 0,C 180,E1 -8661.644,E2 -8661.644} C_VEL
LIN {X 0,Y 446.449,Z 213.876,A -85,B 0,C 180,E1 -8665.153,E2 -8665.153} C_VEL
LIN {X 0,Y 446.49,Z 213.871,A -85,B 0,C 180,E1 -8668.178,E2 -8668.178} C_VEL
LIN {X 0,Y 446.424,Z 213.878,A -85,B 0,C 180,E1 -8671.774,E2 -8671.774} C_VEL
LIN {X 0,Y 446.434,Z 213.876,A -85,B 0,C 180,E1 -8674.523,E2 -8674.523} C_VEL
LIN {X 0,Y 446.421,Z 213.878,A -85,B 0,C 180,E1 -8678.079,E2 -8678.079} C_VEL
LIN {X 0,Y 446.432,Z 213.874,A -85,B 0,C 180,E1 -8680.917,E2 -8680.917} C_VEL
LIN {X 0,Y 446.403,Z 213.88,A -85,B 0,C 180,E1 -8683.846,E2 -8683.846} C_VEL
LIN {X 0,Y 446.403,Z 213.88,A -85,B 0,C 180,E1 -8686.403,E2 -8686.403} C_VEL
LIN {X 0,Y 446.44,Z 213.876,A -85,B 0,C 180,E1 -8689.801,E2 -8689.801} C_VEL
LIN {X 0,Y 446.404,Z 213.879,A -85,B 0,C 180,E1 -8693.254,E2 -8693.254} C_VEL
LIN {X 0,Y 446.453,Z 213.876,A -85,B 0,C 180,E1 -8696.566,E2 -8696.566} C_VEL
LIN {X 0,Y 446.433,Z 213.885,A -85,B 0,C 180,E1 -8699.979,E2 -8699.979} C_VEL
LIN {X 0,Y 446.475,Z 214.018,A -85,B 0,C 180,E1 -8701.768,E2 -8701.768} C_VEL
LIN {X 0,Y 448.949,Z 224.739,A -85,B 0,C 180,E1 -8704.251,E2 -8704.251} C_VEL
LIN {X 0,Y 449.742,Z 229.231,A -85,B 0,C 180,E1 -8705.225,E2 -8705.225} C_VEL
LIN {X 0,Y 448.989,Z 241.527,A -85,B 0,C 180,E1 -8707.601,E2 -8707.601} C_VEL
LIN {X 0,Y 447.736,Z 261.148,A -85,B 0,C 180,E1 -8711.228,E2 -8711.228} C_VEL
LIN {X 0,Y 447.57,Z 264.065,A -85,B 0,C 180,E1 -8711.755,E2 -8711.755} C_VEL
LIN {X 0,Y 450.366,Z 281.039,A -85,B 0,C 180,E1 -8712.285,E2 -8712.285} C_VEL
LIN {X 0,Y 451.179,Z 289.405,A -85,B 0,C 180,E1 -8712.509,E2 -8712.509} C_VEL
LIN {X 0,Y 449.668,Z 375.202,A -85,B 0,C 180,E1 -8714.242,E2 -8714.242} C_VEL
LIN {X 0,Y 449.222,Z 388.667,A -85,B 0,C 180,E1 -8714.691,E2 -8714.691} C_VEL
LIN {X 0,Y 448.645,Z 400.538,A -85,B 0,C 180,E1 -8715.252,E2 -8715.252} C_VEL
LIN {X 0,Y 448.03,Z 413.107,A -85,B 0,C 180,E1 -8716.043,E2 -8716.043} C_VEL
LIN {X 0,Y 447.398,Z 425.013,A -85,B 0,C 180,E1 -8717.001,E2 -8717.001} C_VEL
LIN {X 0,Y 446.903,Z 435.679,A -85,B 0,C 180,E1 -8718.087,E2 -8718.087} C_VEL
LIN {X 0,Y 446.329,Z 445.682,A -85,B 0,C 180,E1 -8719.337,E2 -8719.337} C_VEL
LIN {X 0,Y 445.962,Z 454.427,A -85,B 0,C 180,E1 -8720.703,E2 -8720.703} C_VEL
LIN {X 0,Y 445.698,Z 461.465,A -85,B 0,C 180,E1 -8722.068,E2 -8722.068} C_VEL
